LIN {X 0,Y 361.187,Z 795.351,A -85,B 0,C 180,E1 -13387.357,E2 -13387.357} C_VEL
LIN {X 0,Y 363.65,Z 828.384,A -85,B 0,C 180,E1 -13388.543,E2 -13388.543} C_VEL
LIN {X 0,Y 361.748,Z 885.155,A -85,B 0,C 180,E1 -13390.011,E2 -13390.011} C_VEL
LIN {X 0,Y 361.085,Z 897.459,A -85,B 0,C 180,E1 -13390.491,E2 -13390.491} C_VEL
LIN {X 0,Y 360.263,Z 910.027,A -85,B 0,C 180,E1 -13391.074,E2 -13391.074} C_VEL
LIN {X 0,Y 359.139,Z 922.712,A -85,B 0,C 180,E1 -13391.9,E2 -13391.9} C_VEL
LIN {X 0,Y 357.978,Z 934.051,A -85,B 0,C 180,E1 -13392.872,E2 -13392.872} C_VEL
LIN {X 0,Y 356.772,Z 945.633,A -85,B 0,C 180,E1 -13394.136,E2 -13394.136} C_VEL
LIN {X 0,Y 355.868,Z 954.88,A -85,B 0,C 180,E1 -13395.397,E2 -13395.397} C_VEL
LIN {X 0,Y 355.115,Z 963.565,A -85,B 0,C 180,E1 -13396.843,E2 -13396.843} C_VEL
LIN {X 0,Y 354.408,Z 971.955,A -85,B 0,C 180,E1 -13398.561,E2 -13398.561} C_VEL
LIN {X 0,Y 354.031,Z 978.739,A -85,B 0,C 180,E1 -13400.284,E2 -13400.284} C_VEL
LIN {X 0,Y 353.925,Z 984.165,A -85,B 0,C 180,E1 -13402.008,E2 -13402.008} C_VEL
LIN {X 0,Y 353.966,Z 987.855,A -85,B 0,C 180,E1 -13403.493,E2 -13403.493} C_VEL
LIN {X 0,Y 354.122,Z 991.509,A -85,B 0,C 180,E1 -13405.445,E2 -13405.445} C_VEL
LIN {X 0,Y 354.197,Z 993.033,A -85,B 0,C 180,E1 -13406.586,E2 -13406.586} C_VEL
LIN {X 0,Y 354.246,Z 994.085,A -85,B 0,C 180,E1 -13407.724,E2 -13407.724} C_VEL
LIN {X 0,Y 354.313,Z 994.729,A -85,B 0,C 180,E1 -13408.862,E2 -13408.862} C_VEL
LIN {X 0,Y 354.371,Z 994.965,A -85,B 0,C 180,E1 -13409.998,E2 -13409.998} C_VEL
LIN {X 0,Y 354.307,Z 994.762,A -85,B 0,C 180,E1 -13411.135,E2 -13411.135} C_VEL
LIN {X 0,Y 354.238,Z 994.109,A -85,B 0,C 180,E1 -13412.272,E2 -13412.272} C_VEL
LIN {X 0,Y 354.193,Z 993.052,A -85,B 0,C 180,E1 -13413.411,E2 -13413.411} C_VEL
LIN {X 0,Y 354.116,Z 991.578,A -85,B 0,C 180,E1 -13414.552,E2 -13414.552} C_VEL
LIN {X 0,Y 353.962,Z 987.944,A -85,B 0,C 180,E1 -13416.533,E2 -13416.533} C_VEL
LIN {X 0,Y 353.921,Z 982.715,A -85,B 0,C 180,E1 -13418.563,E2 -13418.563} C_VEL
LIN {X 0,Y 354.153,Z 975.942,A -85,B 0,C 180,E1 -13420.575,E2 -13420.575} C_VEL
LIN {X 0,Y 354.69,Z 968.615,A -85,B 0,C 180,E1 -13422.297,E2 -13422.297} C_VEL
LIN {X 0,Y 355.571,Z 960.085,A -85,B 0,C 180,E1 -13423.915,E2 -13423.915} C_VEL
LIN {X 0,Y 356.435,Z 951.284,A -85,B 0,C 180,E1 -13425.289,E2 -13425.289} C_VEL
LIN {X 0,Y 357.256,Z 942.549,A -85,B 0,C 180,E1 -13426.425,E2 -13426.425} C_VEL
LIN {X 0,Y 358.722,Z 930.579,A -85,B 0,C 180,E1 -13427.676,E2 -13427.676} C_VEL
LIN {X 0,Y 359.936,Z 918.59,A -85,B 0,C 180,E1 -13428.645,E2 -13428.645} C_VEL
LIN {X 0,Y 361.04,Z 906.197,A -85,B 0,C 180,E1 -13429.397,E2 -13429.397} C_VEL
LIN {X 0,Y 361.965,Z 892.632,A -85,B 0,C 180,E1 -13429.973,E2 -13429.973} C_VEL
LIN {X 0,Y 362.399,Z 877.372,A -85,B 0,C 180,E1 -13430.355,E2 -13430.355} C_VEL
LIN {X 0,Y 363.215,Z 826.987,A -85,B 0,C 180,E1 -13431.38,E2 -13431.38} C_VEL
LIN {X 0,Y 359.888,Z 793.813,A -85,B 0,C 180,E1 -13432.316,E2 -13432.316} C_VEL
LIN {X 0,Y 357.689,Z 776.377,A -85,B 0,C 180,E1 -13432.881,E2 -13432.881} C_VEL
LIN {X 0,Y 359.216,Z 759.596,A -85,B 0,C 180,E1 -13435.844,E2 -13435.844} C_VEL
LIN {X 0,Y 361.25,Z 739.879,A -85,B 0,C 180,E1 -13439.419,E2 -13439.419} C_VEL
LIN {X 0,Y 361.354,Z 736.535,A -85,B 0,C 180,E1 -13440.052,E2 -13440.052} C_VEL
LIN {X 0,Y 358.531,Z 723.308,A -85,B 0,C 180,E1 -13442.85,E2 -13442.85} C_VEL
LIN {X 0,Y 355.677,Z 711.544,A -85,B 0,C 180,E1 -13445.502,E2 -13445.502} C_VEL
LIN {X 0,Y 354.855,Z 708.388,A -85,B 0,C 180,E1 -13446.295,E2 -13446.295} C_VEL
LIN {X 0,Y 354.817,Z 708.289,A -85,B 0,C 180,E1 -13449.422,E2 -13449.422} C_VEL
LIN {X 0,Y 354.781,Z 708.286,A -85,B 0,C 180,E1 -13452.866,E2 -13452.866} C_VEL
LIN {X 0,Y 354.761,Z 708.286,A -85,B 0,C 180,E1 -13456.103,E2 -13456.103} C_VEL
LIN {X 0,Y 354.78,Z 708.284,A -85,B 0,C 180,E1 -13459.178,E2 -13459.178} C_VEL
LIN {X 0,Y 354.803,Z 708.289,A -85,B 0,C 180,E1 -13462.4,E2 -13462.4} C_VEL
LIN {X 0,Y 354.802,Z 708.275,A -85,B 0,C 180,E1 -13464.94,E2 -13464.94} C_VEL
LIN {X 0,Y 354.783,Z 708.289,A -85,B 0,C 180,E1 -13468.404,E2 -13468.404} C_VEL
LIN {X 0,Y 354.843,Z 708.281,A -85,B 0,C 180,E1 -13471.618,E2 -13471.618} C_VEL
LIN {X 0,Y 354.888,Z 708.275,A -85,B 0,C 180,E1 -13474.172,E2 -13474.172} C_VEL
LIN {X 0,Y 354.823,Z 708.282,A -85,B 0,C 180,E1 -13477.893,E2 -13477.893} C_VEL
LIN {X 0,Y 354.911,Z 708.27,A -85,B 0,C 180,E1 -13481.891,E2 -13481.891} C_VEL
LIN {X 0,Y 354.931,Z 708.268,A -85,B 0,C 180,E1 -13485.981,E2 -13485.981} C_VEL
LIN {X 0,Y 354.966,Z 708.269,A -85,B 0,C 180,E1 -13489.736,E2 -13489.736} C_VEL
LIN {X 0,Y 355.112,Z 708.248,A -85,B 0,C 180,E1 -13493.18,E2 -13493.18} C_VEL
LIN {X 0,Y 355.234,Z 708.233,A -85,B 0,C 180,E1 -13497.732,E2 -13497.732} C_VEL
LIN {X 0,Y 355.385,Z 708.21,A -85,B 0,C 180,E1 -13500,E2 -13500} C_VEL
LIN {X 0,Y 355.233,Z 708.236,A -85,B 0,C 180,E1 -13502.268,E2 -13502.268} C_VEL
LIN {X 0,Y 355.125,Z 708.249,A -85,B 0,C 180,E1 -13506.82,E2 -13506.82} C_VEL
LIN {X 0,Y 355.004,Z 708.26,A -85,B 0,C 180,E1 -13509.113,E2 -13509.113} C_VEL
LIN {X 0,Y 354.91,Z 708.271,A -85,B 0,C 180,E1 -13512.582,E2 -13512.582} C_VEL
LIN {X 0,Y 354.878,Z 708.272,A -85,B 0,C 180,E1 -13516.097,E2 -13516.097} C_VEL
LIN {X 0,Y 354.89,Z 708.278,A -85,B 0,C 180,E1 -13518.473,E2 -13518.473} C_VEL
LIN {X 0,Y 354.804,Z 708.283,A -85,B 0,C 180,E1 -13522.108,E2 -13522.108} C_VEL
LIN {X 0,Y 354.887,Z 708.281,A -85,B 0,C 180,E1 -13525.829,E2 -13525.829} C_VEL
LIN {X 0,Y 354.808,Z 708.284,A -85,B 0,C 180,E1 -13529.683,E2 -13529.683} C_VEL
LIN {X 0,Y 354.797,Z 708.286,A -85,B 0,C 180,E1 -13533.703,E2 -13533.703} C_VEL
LIN {X 0,Y 354.793,Z 708.285,A -85,B 0,C 180,E1 -13536.461,E2 -13536.461} C_VEL
LIN {X 0,Y 354.816,Z 708.285,A -85,B 0,C 180,E1 -13539.425,E2 -13539.425} C_VEL
LIN {X 0,Y 354.839,Z 708.428,A -85,B 0,C 180,E1 -13542.292,E2 -13542.292} C_VEL
LIN {X 0,Y 355.063,Z 709.428,A -85,B 0,C 180,E1 -13542.499,E2 -13542.499} C_VEL
LIN {X 0,Y 361.993,Z 724.642,A -85,B 0,C 180,E1 -13543.378,E2 -13543.378} C_VEL
LIN {X 0,Y 364.783,Z 731.44,A -85,B 0,C 180,E1 -13543.724,E2 -13543.724} C_VEL
LIN {X 0,Y 363.92,Z 784.743,A -85,B 0,C 180,E1 -13544.825,E2 -13544.825} C_VEL
LIN {X 0,Y 363.875,Z 798.11,A -85,B 0,C 180,E1 -13545.213,E2 -13545.213} C_VEL
LIN {X 0,Y 363.637,Z 810.174,A -85,B 0,C 180,E1 -13545.778,E2 -13545.778} C_VEL
LIN {X 0,Y 363.079,Z 822.796,A -85,B 0,C 180,E1 -13546.597,E2 -13546.597} C_VEL
LIN {X 0,Y 362.232,Z 834.729,A -85,B 0,C 180,E1 -13547.626,E2 -13547.626} C_VEL
LIN {X 0,Y 361.284,Z 845.818,A -85,B 0,C 180,E1 -13548.858,E2 -13548.858} C_VEL
LIN {X 0,Y 360.216,Z 856.083,A -85,B 0,C 180,E1 -13550.288,E2 -13550.288} C_VEL
LIN {X 0,Y 359.068,Z 865.467,A -85,B 0,C 180,E1 -13551.938,E2 -13551.938} C_VEL
LIN {X 0,Y 358.091,Z 872.957,A -85,B 0,C 180,E1 -13553.58,E2 -13553.58} C_VEL
LIN {X 0,Y 357.329,Z 878.96,A -85,B 0,C 180,E1 -13555.226,E2 -13555.226} C_VEL
LIN {X 0,Y 356.46,Z 884.482,A -85,B 0,C 180,E1 -13557.169,E2 -13557.169} C_VEL
LIN {X 0,Y 355.92,Z 888.534,A -85,B 0,C 180,E1 -13559.112,E2 -13559.112} C_VEL
LIN {X 0,Y 355.612,Z 890.545,A -85,B 0,C 180,E1 -13560.41,E2 -13560.41} C_VEL
LIN {X 0,Y 355.379,Z 891.923,A -85,B 0,C 180,E1 -13561.667,E2 -13561.667} C_VEL
LIN {X 0,Y 355.21,Z 892.853,A -85,B 0,C 180,E1 -13562.933,E2 -13562.933} C_VEL
LIN {X 0,Y 355.1,Z 893.271,A -85,B 0,C 180,E1 -13564.19,E2 -13564.19} C_VEL
LIN {X 0,Y 355.01,Z 893.189,A -85,B 0,C 180,E1 -13565.596,E2 -13565.596} C_VEL
LIN {X 0,Y 355.031,Z 892.728,A -85,B 0,C 180,E1 -13566.679,E2 -13566.679} C_VEL
LIN {X 0,Y 355.205,Z 891.198,A -85,B 0,C 180,E1 -13568.425,E2 -13568.425} C_VEL
LIN {X 0,Y 355.566,Z 888.364,A -85,B 0,C 180,E1 -13570.368,E2 -13570.368} C_VEL
LIN {X 0,Y 356.038,Z 884.542,A -85,B 0,C 180,E1 -13572.186,E2 -13572.186} C_VEL
LIN {X 0,Y 356.602,Z 879.534,A -85,B 0,C 180,E1 -13573.985,E2 -13573.985} C_VEL
LIN {X 0,Y 357.322,Z 873.189,A -85,B 0,C 180,E1 -13575.769,E2 -13575.769} C_VEL
LIN {X 0,Y 358.214,Z 865.265,A -85,B 0,C 180,E1 -13577.538,E2 -13577.538} C_VEL
LIN {X 0,Y 359.042,Z 857.126,A -85,B 0,C 180,E1 -13578.999,E2 -13578.999} C_VEL
LIN {X 0,Y 359.999,Z 847.172,A -85,B 0,C 180,E1 -13580.45,E2 -13580.45} C_VEL
LIN {X 0,Y 360.918,Z 836.089,A -85,B 0,C 180,E1 -13581.745,E2 -13581.745} C_VEL
LIN {X 0,Y 361.715,Z 824.779,A -85,B 0,C 180,E1 -13582.779,E2 -13582.779} C_VEL
LIN {X 0,Y 362.31,Z 812.227,A -85,B 0,C 180,E1 -13583.668,E2 -13583.668} C_VEL
LIN {X 0,Y 362.675,Z 799.879,A -85,B 0,C 180,E1 -13584.302,E2 -13584.302} C_VEL
LIN {X 0,Y 362.785,Z 787.742,A -85,B 0,C 180,E1 -13584.717,E2 -13584.717} C_VEL
LIN {X 0,Y 363.57,Z 731.522,A -85,B 0,C 180,E1 -13585.873,E2 -13585.873} C_VEL
LIN {X 0,Y 363.342,Z 729.011,A -85,B 0,C 180,E1 -13585.94,E2 -13585.94} C_VEL
LIN {X 0,Y 355.205,Z 709.198,A -85,B 0,C 180,E1 -13586.883,E2 -13586.883} C_VEL
LIN {X 0,Y 355.09,Z 708.341,A -85,B 0,C 180,E1 -13587.095,E2 -13587.095} C_VEL
LIN {X 0,Y 355.148,Z 708.249,A -85,B 0,C 180,E1 -13588.868,E2 -13588.868} C_VEL
LIN {X 0,Y 355.222,Z 708.236,A -85,B 0,C 180,E1 -13592.269,E2 -13592.269} C_VEL
LIN {X 0,Y 355.089,Z 708.249,A -85,B 0,C 180,E1 -13596.822,E2 -13596.822} C_VEL
LIN {X 0,Y 354.955,Z 708.265,A -85,B 0,C 180,E1 -13600.266,E2 -13600.266} C_VEL
LIN {X 0,Y 354.948,Z 708.267,A -85,B 0,C 180,E1 -13604.02,E2 -13604.02} C_VEL
LIN {X 0,Y 354.872,Z 708.279,A -85,B 0,C 180,E1 -13607.518,E2 -13607.518} C_VEL
LIN {X 0,Y 354.823,Z 708.283,A -85,B 0,C 180,E1 -13611.418,E2 -13611.418} C_VEL
LIN {X 0,Y 354.794,Z 708.285,A -85,B 0,C 180,E1 -13612.45,E2 -13612.45} C_VEL
LIN {X 0,Y 354.118,Z 708.375,A -85,B 0,C 180,E1 -13613.396,E2 -13613.396} C_VEL
LIN {X 0,Y 351.283,Z 708.719,A -85,B 0,C 180,E1 -13614.937,E2 -13614.937} C_VEL
LIN {X 0,Y 348.879,Z 709.01,A -85,B 0,C 180,E1 -13616.183,E2 -13616.183} C_VEL
LIN {X 0,Y 347.832,Z 709.14,A -85,B 0,C 180,E1 -13617.147,E2 -13617.147} C_VEL
LIN {X 0,Y 347.738,Z 709.155,A -85,B 0,C 180,E1 -13617.473,E2 -13617.473} C_VEL
LIN {X 0,Y 347.736,Z 709.167,A -85,B 0,C 180,E1 -13620.351,E2 -13620.351} C_VEL
LIN {X 0,Y 347.755,Z 709.143,A -85,B 0,C 180,E1 -13624.045,E2 -13624.045} C_VEL
LIN {X 0,Y 347.76,Z 709.155,A -85,B 0,C 180,E1 -13627.323,E2 -13627.323} C_VEL
LIN {X 0,Y 347.702,Z 709.171,A -85,B 0,C 180,E1 -13630.303,E2 -13630.303} C_VEL
LIN {X 0,Y 347.72,Z 709.173,A -85,B 0,C 180,E1 -13633.411,E2 -13633.411} C_VEL
LIN {X 0,Y 347.728,Z 709.168,A -85,B 0,C 180,E1 -13636.688,E2 -13636.688} C_VEL
LIN {X 0,Y 347.708,Z 709.174,A -85,B 0,C 180,E1 -13640.183,E2 -13640.183} C_VEL
LIN {X 0,Y 347.76,Z 709.166,A -85,B 0,C 180,E1 -13642.678,E2 -13642.678} C_VEL
LIN {X 0,Y 347.857,Z 709.393,A -85,B 0,C 180,E1 -13645.736,E2 -13645.736} C_VEL
LIN {X 0,Y 348.03,Z 710.197,A -85,B 0,C 180,E1 -13645.89,E2 -13645.89} C_VEL
LIN {X 0,Y 354.796,Z 729.357,A -85,B 0,C 180,E1 -13646.733,E2 -13646.733} C_VEL
LIN {X 0,Y 353.601,Z 786.373,A -85,B 0,C 180,E1 -13648.146,E2 -13648.146} C_VEL
LIN {X 0,Y 353.411,Z 797.802,A -85,B 0,C 180,E1 -13648.596,E2 -13648.596} C_VEL
LIN {X 0,Y 353.102,Z 808.375,A -85,B 0,C 180,E1 -13649.168,E2 -13649.168} C_VEL
LIN {X 0,Y 352.703,Z 817.545,A -85,B 0,C 180,E1 -13649.792,E2 -13649.792} C_VEL
LIN {X 0,Y 352.091,Z 828.422,A -85,B 0,C 180,E1 -13650.722,E2 -13650.722} C_VEL
LIN {X 0,Y 351.487,Z 837.924,A -85,B 0,C 180,E1 -13651.72,E2 -13651.72} C_VEL
LIN {X 0,Y 350.886,Z 846.039,A -85,B 0,C 180,E1 -13652.731,E2 -13652.731} C_VEL
LIN {X 0,Y 350.414,Z 853.461,A -85,B 0,C 180,E1 -13653.817,E2 -13653.817} C_VEL
LIN {X 0,Y 349.887,Z 860.653,A -85,B 0,C 180,E1 -13655.05,E2 -13655.05} C_VEL
LIN {X 0,Y 349.234,Z 868.074,A -85,B 0,C 180,E1 -13656.581,E2 -13656.581} C_VEL
LIN {X 0,Y 348.791,Z 873.676,A -85,B 0,C 180,E1 -13657.957,E2 -13657.957} C_VEL
LIN {X 0,Y 348.471,Z 878.376,A -85,B 0,C 180,E1 -13659.332,E2 -13659.332} C_VEL
LIN {X 0,Y 348.153,Z 883.303,A -85,B 0,C 180,E1 -13661.156,E2 -13661.156} C_VEL
LIN {X 0,Y 347.914,Z 886.997,A -85,B 0,C 180,E1 -13662.968,E2 -13662.968} C_VEL
LIN {X 0,Y 347.775,Z 889.586,A -85,B 0,C 180,E1 -13664.769,E2 -13664.769} C_VEL
LIN {X 0,Y 347.82,Z 890.797,A -85,B 0,C 180,E1 -13665.967,E2 -13665.967} C_VEL
LIN {X 0,Y 347.854,Z 891.478,A -85,B 0,C 180,E1 -13667.159,E2 -13667.159} C_VEL
LIN {X 0,Y 347.981,Z 891.721,A -85,B 0,C 180,E1 -13668.348,E2 -13668.348} C_VEL
LIN {X 0,Y 348.178,Z 891.547,A -85,B 0,C 180,E1 -13669.533,E2 -13669.533} C_VEL
LIN {X 0,Y 348.509,Z 890.537,A -85,B 0,C 180,E1 -13671.172,E2 -13671.172} C_VEL
LIN {X 0,Y 349.011,Z 888.328,A -85,B 0,C 180,E1 -13673.06,E2 -13673.06} C_VEL
LIN {X 0,Y 349.623,Z 885.176,A -85,B 0,C 180,E1 -13674.81,E2 -13674.81} C_VEL
LIN {X 0,Y 350.327,Z 880.893,A -85,B 0,C 180,E1 -13676.549,E2 -13676.549} C_VEL
LIN {X 0,Y 351.132,Z 875.354,A -85,B 0,C 180,E1 -13678.279,E2 -13678.279} C_VEL
LIN {X 0,Y 352.021,Z 870.096,A -85,B 0,C 180,E1 -13679.62,E2 -13679.62} C_VEL
LIN {X 0,Y 353.034,Z 862.825,A -85,B 0,C 180,E1 -13681.141,E2 -13681.141} C_VEL
LIN {X 0,Y 353.898,Z 856.366,A -85,B 0,C 180,E1 -13682.276,E2 -13682.276} C_VEL
LIN {X 0,Y 354.886,Z 847.639,A -85,B 0,C 180,E1 -13683.548,E2 -13683.548} C_VEL
LIN {X 0,Y 355.855,Z 838.207,A -85,B 0,C 180,E1 -13684.673,E2 -13684.673} C_VEL
LIN {X 0,Y 356.553,Z 829.764,A -85,B 0,C 180,E1 -13685.514,E2 -13685.514} C_VEL
LIN {X 0,Y 357.209,Z 819.421,A -85,B 0,C 180,E1 -13686.354,E2 -13686.354} C_VEL
LIN {X 0,Y 357.742,Z 809.048,A -85,B 0,C 180,E1 -13687.017,E2 -13687.017} C_VEL
LIN {X 0,Y 358.112,Z 798.99,A -85,B 0,C 180,E1 -13687.506,E2 -13687.506} C_VEL
LIN {X 0,Y 358.317,Z 785.894,A -85,B 0,C 180,E1 -13687.959,E2 -13687.959} C_VEL
LIN {X 0,Y 359.291,Z 754.548,A -85,B 0,C 180,E1 -13688.813,E2 -13688.813} C_VEL
LIN {X 0,Y 360.134,Z 733.434,A -85,B 0,C 180,E1 -13689.39,E2 -13689.39} C_VEL
LIN {X 0,Y 354.89,Z 722.496,A -85,B 0,C 180,E1 -13690.29,E2 -13690.29} C_VEL
LIN {X 0,Y 349.346,Z 712.616,A -85,B 0,C 180,E1 -13691.263,E2 -13691.263} C_VEL
LIN {X 0,Y 347.986,Z 709.706,A -85,B 0,C 180,E1 -13691.585,E2 -13691.585} C_VEL
LIN {X 0,Y 347.883,Z 709.168,A -85,B 0,C 180,E1 -13691.951,E2 -13691.951} C_VEL
LIN {X 0,Y 347.872,Z 709.153,A -85,B 0,C 180,E1 -13695.226,E2 -13695.226} C_VEL
LIN {X 0,Y 347.81,Z 709.161,A -85,B 0,C 180,E1 -13698.863,E2 -13698.863} C_VEL
LIN {X 0,Y 347.769,Z 709.168,A -85,B 0,C 180,E1 -13702.58,E2 -13702.58} C_VEL
LIN {X 0,Y 347.8,Z 709.161,A -85,B 0,C 180,E1 -13705.109,E2 -13705.109} C_VEL
LIN {X 0,Y 347.764,Z 709.166,A -85,B 0,C 180,E1 -13709.014,E2 -13709.014} C_VEL
LIN {X 0,Y 347.74,Z 709.17,A -85,B 0,C 180,E1 -13713.071,E2 -13713.071} C_VEL
LIN {X 0,Y 347.777,Z 709.164,A -85,B 0,C 180,E1 -13716.064,E2 -13716.064} C_VEL
LIN {X 0,Y 347.759,Z 709.165,A -85,B 0,C 180,E1 -13718.792,E2 -13718.792} C_VEL
LIN {X 0,Y 347.757,Z 709.168,A -85,B 0,C 180,E1 -13721.829,E2 -13721.829} C_VEL
LIN {X 0,Y 347.712,Z 709.171,A -85,B 0,C 180,E1 -13725.026,E2 -13725.026} C_VEL
LIN {X 0,Y 347.756,Z 709.167,A -85,B 0,C 180,E1 -13728.396,E2 -13728.396} C_VEL
LIN {X 0,Y 347.778,Z 709.165,A -85,B 0,C 180,E1 -13732.01,E2 -13732.01} C_VEL
LIN {X 0,Y 347.815,Z 709.357,A -85,B 0,C 180,E1 -13733.781,E2 -13733.781} C_VEL
LIN {X 0,Y 351.296,Z 723.703,A -85,B 0,C 180,E1 -13736.963,E2 -13736.963} C_VEL
LIN {X 0,Y 354.079,Z 736.282,A -85,B 0,C 180,E1 -13739.591,E2 -13739.591} C_VEL
LIN {X 0,Y 354.337,Z 739.773,A -85,B 0,C 180,E1 -13740.272,E2 -13740.272} C_VEL
LIN {X 0,Y 352.046,Z 761.67,A -85,B 0,C 180,E1 -13744.264,E2 -13744.264} C_VEL
LIN {X 0,Y 351.359,Z 769.237,A -85,B 0,C 180,E1 -13745.572,E2 -13745.572} C_VEL
LIN {X 0,Y 354.075,Z 789.134,A -85,B 0,C 180,E1 -13746.512,E2 -13746.512} C_VEL
LIN {X 0,Y 355.43,Z 801.877,A -85,B 0,C 180,E1 -13747.047,E2 -13747.047} C_VEL
LIN {X 0,Y 357.266,Z 829.438,A -85,B 0,C 180,E1 -13748.051,E2 -13748.051} C_VEL
LIN {X 0,Y 355.318,Z 884.018,A -85,B 0,C 180,E1 -13749.52,E2 -13749.52} C_VEL
LIN {X 0,Y 354.697,Z 894.667,A -85,B 0,C 180,E1 -13749.937,E2 -13749.937} C_VEL
LIN {X 0,Y 353.755,Z 906.444,A -85,B 0,C 180,E1 -13750.561,E2 -13750.561} C_VEL
LIN {X 0,Y 352.389,Z 921.354,A -85,B 0,C 180,E1 -13751.54,E2 -13751.54} C_VEL
LIN {X 0,Y 351.173,Z 932.777,A -85,B 0,C 180,E1 -13752.529,E2 -13752.529} C_VEL
LIN {X 0,Y 350.055,Z 943.219,A -85,B 0,C 180,E1 -13753.674,E2 -13753.674} C_VEL
LIN {X 0,Y 349.023,Z 953.3,A -85,B 0,C 180,E1 -13755.043,E2 -13755.043} C_VEL
LIN {X 0,Y 348.18,Z 962.42,A -85,B 0,C 180,E1 -13756.576,E2 -13756.576} C_VEL
LIN {X 0,Y 347.404,Z 970.83,A -85,B 0,C 180,E1 -13758.327,E2 -13758.327} C_VEL
LIN {X 0,Y 346.999,Z 977.635,A -85,B 0,C 180,E1 -13760.085,E2 -13760.085} C_VEL
LIN {X 0,Y 346.862,Z 983.078,A -85,B 0,C 180,E1 -13761.844,E2 -13761.844} C_VEL
LIN {X 0,Y 346.919,Z 986.997,A -85,B 0,C 180,E1 -13763.454,E2 -13763.454} C_VEL
LIN {X 0,Y 347.062,Z 990.46,A -85,B 0,C 180,E1 -13765.352,E2 -13765.352} C_VEL
LIN {X 0,Y 347.152,Z 991.999,A -85,B 0,C 180,E1 -13766.516,E2 -13766.516} C_VEL
LIN {X 0,Y 347.205,Z 993.06,A -85,B 0,C 180,E1 -13767.678,E2 -13767.678} C_VEL
LIN {X 0,Y 347.279,Z 993.711,A -85,B 0,C 180,E1 -13768.839,E2 -13768.839} C_VEL
LIN {X 0,Y 347.343,Z 993.953,A -85,B 0,C 180,E1 -13769.998,E2 -13769.998} C_VEL
LIN {X 0,Y 347.271,Z 993.758,A -85,B 0,C 180,E1 -13771.158,E2 -13771.158} C_VEL
LIN {X 0,Y 347.195,Z 993.11,A -85,B 0,C 180,E1 -13772.318,E2 -13772.318} C_VEL
LIN {X 0,Y 347.148,Z 992.057,A -85,B 0,C 180,E1 -13773.48,E2 -13773.48} C_VEL
LIN {X 0,Y 347.056,Z 990.583,A -85,B 0,C 180,E1 -13774.644,E2 -13774.644} C_VEL
LIN {X 0,Y 346.919,Z 987.211,A -85,B 0,C 180,E1 -13776.546,E2 -13776.546} C_VEL
LIN {X 0,Y 346.833,Z 983.37,A -85,B 0,C 180,E1 -13778.153,E2 -13778.153} C_VEL
LIN {X 0,Y 347.009,Z 977.097,A -85,B 0,C 180,E1 -13780.206,E2 -13780.206} C_VEL
LIN {X 0,Y 347.493,Z 970.264,A -85,B 0,C 180,E1 -13781.963,E2 -13781.963} C_VEL
LIN {X 0,Y 348.159,Z 963.381,A -85,B 0,C 180,E1 -13783.421,E2 -13783.421} C_VEL
LIN {X 0,Y 349.045,Z 954.52,A -85,B 0,C 180,E1 -13784.972,E2 -13784.972} C_VEL
LIN {X 0,Y 350.158,Z 944.035,A -85,B 0,C 180,E1 -13786.467,E2 -13786.467} C_VEL
LIN {X 0,Y 351.575,Z 932.67,A -85,B 0,C 180,E1 -13787.747,E2 -13787.747} C_VEL
LIN {X 0,Y 352.811,Z 921.592,A -85,B 0,C 180,E1 -13788.734,E2 -13788.734} C_VEL
LIN {X 0,Y 354.056,Z 909.409,A -85,B 0,C 180,E1 -13789.569,E2 -13789.569} C_VEL
LIN {X 0,Y 355.016,Z 896.926,A -85,B 0,C 180,E1 -13790.192,E2 -13790.192} C_VEL
LIN {X 0,Y 355.654,Z 884.128,A -85,B 0,C 180,E1 -13790.607,E2 -13790.607} C_VEL
LIN {X 0,Y 356.612,Z 827.527,A -85,B 0,C 180,E1 -13791.794,E2 -13791.794} C_VEL
LIN {X 0,Y 353.362,Z 794.632,A -85,B 0,C 180,E1 -13792.743,E2 -13792.743} C_VEL
LIN {X 0,Y 350.889,Z 775.382,A -85,B 0,C 180,E1 -13793.376,E2 -13793.376} C_VEL
LIN {X 0,Y 352.424,Z 759.116,A -85,B 0,C 180,E1 -13796.306,E2 -13796.306} C_VEL
LIN {X 0,Y 354.45,Z 740.741,A -85,B 0,C 180,E1 -13799.714,E2 -13799.714} C_VEL
LIN {X 0,Y 354.373,Z 737.386,A -85,B 0,C 180,E1 -13800.377,E2 -13800.377} C_VEL
LIN {X 0,Y 351.589,Z 724.466,A -85,B 0,C 180,E1 -13803.186,E2 -13803.186} C_VEL
LIN {X 0,Y 348.899,Z 713.443,A -85,B 0,C 180,E1 -13805.741,E2 -13805.741} C_VEL
LIN {X 0,Y 347.799,Z 709.247,A -85,B 0,C 180,E1 -13806.824,E2 -13806.824} C_VEL
LIN {X 0,Y 347.725,Z 709.167,A -85,B 0,C 180,E1 -13810.295,E2 -13810.295} C_VEL
LIN {X 0,Y 347.719,Z 709.166,A -85,B 0,C 180,E1 -13813.406,E2 -13813.406} C_VEL
LIN {X 0,Y 347.717,Z 709.164,A -85,B 0,C 180,E1 -13816.685,E2 -13816.685} C_VEL
LIN {X 0,Y 347.738,Z 709.156,A -85,B 0,C 180,E1 -13820.172,E2 -13820.172} C_VEL
LIN {X 0,Y 347.756,Z 709.169,A -85,B 0,C 180,E1 -13822.679,E2 -13822.679} C_VEL
LIN {X 0,Y 347.738,Z 709.165,A -85,B 0,C 180,E1 -13825.955,E2 -13825.955} C_VEL
LIN {X 0,Y 347.754,Z 709.169,A -85,B 0,C 180,E1 -13829.653,E2 -13829.653} C_VEL
LIN {X 0,Y 347.842,Z 709.153,A -85,B 0,C 180,E1 -13832.743,E2 -13832.743} C_VEL
LIN {X 0,Y 347.777,Z 709.163,A -85,B 0,C 180,E1 -13836.161,E2 -13836.161} C_VEL
LIN {X 0,Y 347.806,Z 709.161,A -85,B 0,C 180,E1 -13839.909,E2 -13839.909} C_VEL
LIN {X 0,Y 347.855,Z 709.146,A -85,B 0,C 180,E1 -13842.359,E2 -13842.359} C_VEL
LIN {X 0,Y 347.885,Z 709.145,A -85,B 0,C 180,E1 -13845.97,E2 -13845.97} C_VEL
LIN {X 0,Y 347.916,Z 709.147,A -85,B 0,C 180,E1 -13849.525,E2 -13849.525} C_VEL
LIN {X 0,Y 348.078,Z 709.125,A -85,B 0,C 180,E1 -13853.042,E2 -13853.042} C_VEL
LIN {X 0,Y 348.197,Z 709.109,A -85,B 0,C 180,E1 -13857.687,E2 -13857.687} C_VEL
LIN {X 0,Y 348.334,Z 709.088,A -85,B 0,C 180,E1 -13860,E2 -13860} C_VEL
LIN {X 0,Y 348.196,Z 709.113,A -85,B 0,C 180,E1 -13862.314,E2 -13862.314} C_VEL
LIN {X 0,Y 348.093,Z 709.124,A -85,B 0,C 180,E1 -13866.958,E2 -13866.958} C_VEL
LIN {X 0,Y 347.956,Z 709.139,A -85,B 0,C 180,E1 -13869.299,E2 -13869.299} C_VEL
LIN {X 0,Y 347.879,Z 709.147,A -85,B 0,C 180,E1 -13872.84,E2 -13872.84} C_VEL
LIN {X 0,Y 347.827,Z 709.151,A -85,B 0,C 180,E1 -13876.432,E2 -13876.432} C_VEL
LIN {X 0,Y 347.839,Z 709.154,A -85,B 0,C 180,E1 -13878.861,E2 -13878.861} C_VEL
LIN {X 0,Y 347.751,Z 709.156,A -85,B 0,C 180,E1 -13882.581,E2 -13882.581} C_VEL
LIN {X 0,Y 347.8,Z 709.155,A -85,B 0,C 180,E1 -13885.11,E2 -13885.11} C_VEL
LIN {X 0,Y 347.798,Z 709.152,A -85,B 0,C 180,E1 -13887.695,E2 -13887.695} C_VEL
LIN {X 0,Y 347.74,Z 709.171,A -85,B 0,C 180,E1 -13890.349,E2 -13890.349} C_VEL
LIN {X 0,Y 347.739,Z 709.17,A -85,B 0,C 180,E1 -13894.045,E2 -13894.045} C_VEL
LIN {X 0,Y 347.758,Z 709.168,A -85,B 0,C 180,E1 -13897.322,E2 -13897.322} C_VEL
LIN {X 0,Y 347.725,Z 709.172,A -85,B 0,C 180,E1 -13900.298,E2 -13900.298} C_VEL
LIN {X 0,Y 347.786,Z 709.337,A -85,B 0,C 180,E1 -13901.769,E2 -13901.769} C_VEL
LIN {X 0,Y 348.057,Z 710.428,A -85,B 0,C 180,E1 -13901.98,E2 -13901.98} C_VEL
LIN {X 0,Y 355.106,Z 725.654,A -85,B 0,C 180,E1 -13902.897,E2 -13902.897} C_VEL
LIN {X 0,Y 358.261,Z 732.986,A -85,B 0,C 180,E1 -13903.294,E2 -13903.294} C_VEL
LIN {X 0,Y 357.367,Z 788.959,A -85,B 0,C 180,E1 -13904.483,E2 -13904.483} C_VEL
LIN {X 0,Y 357.262,Z 802.328,A -85,B 0,C 180,E1 -13904.935,E2 -13904.935} C_VEL
LIN {X 0,Y 356.958,Z 814.44,A -85,B 0,C 180,E1 -13905.566,E2 -13905.566} C_VEL
LIN {X 0,Y 356.365,Z 825.612,A -85,B 0,C 180,E1 -13906.353,E2 -13906.353} C_VEL
LIN {X 0,Y 355.424,Z 837.818,A -85,B 0,C 180,E1 -13907.475,E2 -13907.475} C_VEL
LIN {X 0,Y 354.457,Z 848.554,A -85,B 0,C 180,E1 -13908.736,E2 -13908.736} C_VEL
LIN {X 0,Y 353.214,Z 858.923,A -85,B 0,C 180,E1 -13910.27,E2 -13910.27} C_VEL
LIN {X 0,Y 352.198,Z 867.163,A -85,B 0,C 180,E1 -13911.789,E2 -13911.789} C_VEL
LIN {X 0,Y 351.178,Z 874.548,A -85,B 0,C 180,E1 -13913.467,E2 -13913.467} C_VEL
LIN {X 0,Y 350.245,Z 881.069,A -85,B 0,C 180,E1 -13915.357,E2 -13915.357} C_VEL
LIN {X 0,Y 349.473,Z 885.814,A -85,B 0,C 180,E1 -13917.116,E2 -13917.116} C_VEL
LIN {X 0,Y 348.921,Z 889.783,A -85,B 0,C 180,E1 -13919.097,E2 -13919.097} C_VEL
LIN {X 0,Y 348.48,Z 892.453,A -85,B 0,C 180,E1 -13921.054,E2 -13921.054} C_VEL
LIN {X 0,Y 348.239,Z 893.721,A -85,B 0,C 180,E1 -13922.622,E2 -13922.622} C_VEL
LIN {X 0,Y 348.033,Z 894.328,A -85,B 0,C 180,E1 -13924.911,E2 -13924.911} C_VEL
LIN {X 0,Y 347.982,Z 893.979,A -85,B 0,C 180,E1 -13926.178,E2 -13926.178} C_VEL
LIN {X 0,Y 348.171,Z 892.462,A -85,B 0,C 180,E1 -13928.208,E2 -13928.208} C_VEL
LIN {X 0,Y 348.589,Z 889.135,A -85,B 0,C 180,E1 -13930.572,E2 -13930.572} C_VEL
LIN {X 0,Y 349.076,Z 885.239,A -85,B 0,C 180,E1 -13932.424,E2 -13932.424} C_VEL
LIN {X 0,Y 349.7,Z 880.201,A -85,B 0,C 180,E1 -13934.24,E2 -13934.24} C_VEL
LIN {X 0,Y 350.463,Z 873.704,A -85,B 0,C 180,E1 -13936.077,E2 -13936.077} C_VEL
LIN {X 0,Y 351.244,Z 866.967,A -85,B 0,C 180,E1 -13937.61,E2 -13937.61} C_VEL
LIN {X 0,Y 352.092,Z 859.175,A -85,B 0,C 180,E1 -13939.071,E2 -13939.071} C_VEL
LIN {X 0,Y 353.068,Z 849.448,A -85,B 0,C 180,E1 -13940.55,E2 -13940.55} C_VEL
LIN {X 0,Y 354.023,Z 838.649,A -85,B 0,C 180,E1 -13941.87,E2 -13941.87} C_VEL
LIN {X 0,Y 354.844,Z 828.02,A -85,B 0,C 180,E1 -13942.908,E2 -13942.908} C_VEL
LIN {X 0,Y 355.498,Z 815.85,A -85,B 0,C 180,E1 -13943.831,E2 -13943.831} C_VEL
LIN {X 0,Y 355.915,Z 802.681,A -85,B 0,C 180,E1 -13944.566,E2 -13944.566} C_VEL
LIN {X 0,Y 356.105,Z 790.325,A -85,B 0,C 180,E1 -13945.029,E2 -13945.029} C_VEL
LIN {X 0,Y 356.606,Z 744.348,A -85,B 0,C 180,E1 -13946.012,E2 -13946.012} C_VEL
LIN {X 0,Y 356.74,Z 730.81,A -85,B 0,C 180,E1 -13946.297,E2 -13946.297} C_VEL
LIN {X 0,Y 348.227,Z 709.924,A -85,B 0,C 180,E1 -13947.327,E2 -13947.327} C_VEL
LIN {X 0,Y 348.15,Z 709.187,A -85,B 0,C 180,E1 -13947.543,E2 -13947.543} C_VEL
LIN {X 0,Y 348.12,Z 709.122,A -85,B 0,C 180,E1 -13951.159,E2 -13951.159} C_VEL
LIN {X 0,Y 348.184,Z 709.112,A -85,B 0,C 180,E1 -13952.315,E2 -13952.315} C_VEL
LIN {X 0,Y 348.057,Z 709.124,A -85,B 0,C 180,E1 -13956.96,E2 -13956.96} C_VEL
LIN {X 0,Y 347.895,Z 709.144,A -85,B 0,C 180,E1 -13960.477,E2 -13960.477} C_VEL
LIN {X 0,Y 347.905,Z 709.143,A -85,B 0,C 180,E1 -13964.151,E2 -13964.151} C_VEL
LIN {X 0,Y 347.836,Z 709.155,A -85,B 0,C 180,E1 -13967.644,E2 -13967.644} C_VEL
LIN {X 0,Y 347.77,Z 709.162,A -85,B 0,C 180,E1 -13971.626,E2 -13971.626} C_VEL
LIN {X 0,Y 347.744,Z 709.157,A -85,B 0,C 180,E1 -13975.115,E2 -13975.115} C_VEL
LIN {X 0,Y 347.738,Z 709.155,A -85,B 0,C 180,E1 -13977.473,E2 -13977.473} C_VEL
LIN {X 0,Y 347.054,Z 709.251,A -85,B 0,C 180,E1 -13978.44,E2 -13978.44} C_VEL
LIN {X 0,Y 344.219,Z 709.616,A -85,B 0,C 180,E1 -13980.013,E2 -13980.013} C_VEL
LIN {X 0,Y 341.819,Z 709.913,A -85,B 0,C 180,E1 -13981.286,E2 -13981.286} C_VEL
LIN {X 0,Y 340.773,Z 710.032,A -85,B 0,C 180,E1 -13982.27,E2 -13982.27} C_VEL
LIN {X 0,Y 340.678,Z 710.038,A -85,B 0,C 180,E1 -13982.604,E2 -13982.604} C_VEL
LIN {X 0,Y 340.722,Z 710.016,A -85,B 0,C 180,E1 -13985.28,E2 -13985.28} C_VEL
LIN {X 0,Y 340.699,Z 710.041,A -85,B 0,C 180,E1 -13988.383,E2 -13988.383} C_VEL
LIN {X 0,Y 340.671,Z 710.049,A -85,B 0,C 180,E1 -13992.04,E2 -13992.04} C_VEL
LIN {X 0,Y 340.637,Z 710.056,A -85,B 0,C 180,E1 -13995.453,E2 -13995.453} C_VEL
LIN {X 0,Y 340.675,Z 710.047,A -85,B 0,C 180,E1 -13998.688,E2 -13998.688} C_VEL
LIN {X 0,Y 340.724,Z 710.044,A -85,B 0,C 180,E1 -14001.771,E2 -14001.771} C_VEL
LIN {X 0,Y 340.774,Z 710.195,A -85,B 0,C 180,E1 -14005.374,E2 -14005.374} C_VEL
LIN {X 0,Y 340.999,Z 711.108,A -85,B 0,C 180,E1 -14005.568,E2 -14005.568} C_VEL
LIN {X 0,Y 347.987,Z 730.963,A -85,B 0,C 180,E1 -14006.459,E2 -14006.459} C_VEL
LIN {X 0,Y 346.754,Z 786.436,A -85,B 0,C 180,E1 -14007.857,E2 -14007.857} C_VEL
LIN {X 0,Y 346.533,Z 798.8,A -85,B 0,C 180,E1 -14008.351,E2 -14008.351} C_VEL
LIN {X 0,Y 346.187,Z 809.675,A -85,B 0,C 180,E1 -14008.955,E2 -14008.955} C_VEL
LIN {X 0,Y 345.745,Z 819.212,A -85,B 0,C 180,E1 -14009.626,E2 -14009.626} C_VEL
LIN {X 0,Y 345.1,Z 829.968,A -85,B 0,C 180,E1 -14010.573,E2 -14010.573} C_VEL
LIN {X 0,Y 344.526,Z 839.112,A -85,B 0,C 180,E1 -14011.558,E2 -14011.558} C_VEL
LIN {X 0,Y 343.885,Z 847.449,A -85,B 0,C 180,E1 -14012.623,E2 -14012.623} C_VEL
LIN {X 0,Y 343.351,Z 855.582,A -85,B 0,C 180,E1 -14013.862,E2 -14013.862} C_VEL
LIN {X 0,Y 342.782,Z 862.731,A -85,B 0,C 180,E1 -14015.146,E2 -14015.146} C_VEL
LIN {X 0,Y 342.267,Z 868.704,A -85,B 0,C 180,E1 -14016.396,E2 -14016.396} C_VEL
LIN {X 0,Y 341.846,Z 874.008,A -85,B 0,C 180,E1 -14017.695,E2 -14017.695} C_VEL
LIN {X 0,Y 341.396,Z 880.015,A -85,B 0,C 180,E1 -14019.515,E2 -14019.515} C_VEL
LIN {X 0,Y 341.194,Z 883.416,A -85,B 0,C 180,E1 -14020.757,E2 -14020.757} C_VEL
LIN {X 0,Y 340.952,Z 887.417,A -85,B 0,C 180,E1 -14022.609,E2 -14022.609} C_VEL
LIN {X 0,Y 340.769,Z 890.259,A -85,B 0,C 180,E1 -14024.448,E2 -14024.448} C_VEL
LIN {X 0,Y 340.82,Z 892.41,A -85,B 0,C 180,E1 -14026.889,E2 -14026.889} C_VEL
LIN {X 0,Y 340.937,Z 892.808,A -85,B 0,C 180,E1 -14028.104,E2 -14028.104} C_VEL
LIN {X 0,Y 341.133,Z 892.748,A -85,B 0,C 180,E1 -14029.314,E2 -14029.314} C_VEL
LIN {X 0,Y 341.668,Z 891.332,A -85,B 0,C 180,E1 -14031.721,E2 -14031.721} C_VEL
LIN {X 0,Y 341.979,Z 889.938,A -85,B 0,C 180,E1 -14032.917,E2 -14032.917} C_VEL
LIN {X 0,Y 342.873,Z 885.817,A -85,B 0,C 180,E1 -14035.297,E2 -14035.297} C_VEL
LIN {X 0,Y 343.643,Z 881.42,A -85,B 0,C 180,E1 -14037.069,E2 -14037.069} C_VEL
LIN {X 0,Y 344.473,Z 876.355,A -85,B 0,C 180,E1 -14038.67,E2 -14038.67} C_VEL
LIN {X 0,Y 345.386,Z 871.216,A -85,B 0,C 180,E1 -14040,E2 -14040} C_VEL
LIN {X 0,Y 346.388,Z 864.437,A -85,B 0,C 180,E1 -14041.453,E2 -14041.453} C_VEL
LIN {X 0,Y 347.51,Z 856.18,A -85,B 0,C 180,E1 -14042.898,E2 -14042.898} C_VEL
LIN {X 0,Y 348.48,Z 848.309,A -85,B 0,C 180,E1 -14044.048,E2 -14044.048} C_VEL
LIN {X 0,Y 349.379,Z 840.176,A -85,B 0,C 180,E1 -14045.049,E2 -14045.049} C_VEL
LIN {X 0,Y 350.271,Z 830.335,A -85,B 0,C 180,E1 -14046.047,E2 -14046.047} C_VEL
LIN {X 0,Y 350.876,Z 821.88,A -85,B 0,C 180,E1 -14046.758,E2 -14046.758} C_VEL
LIN {X 0,Y 351.486,Z 811.204,A -85,B 0,C 180,E1 -14047.468,E2 -14047.468} C_VEL
LIN {X 0,Y 351.874,Z 800.678,A -85,B 0,C 180,E1 -14048.001,E2 -14048.001} C_VEL
LIN {X 0,Y 352.075,Z 788.113,A -85,B 0,C 180,E1 -14048.456,E2 -14048.456} C_VEL
LIN {X 0,Y 352.824,Z 764.498,A -85,B 0,C 180,E1 -14049.123,E2 -14049.123} C_VEL
LIN {X 0,Y 354.013,Z 735.573,A -85,B 0,C 180,E1 -14049.944,E2 -14049.944} C_VEL
LIN {X 0,Y 348.243,Z 723.848,A -85,B 0,C 180,E1 -14050.98,E2 -14050.98} C_VEL
LIN {X 0,Y 342.629,Z 713.931,A -85,B 0,C 180,E1 -14052.034,E2 -14052.034} C_VEL
LIN {X 0,Y 341.061,Z 711.072,A -85,B 0,C 180,E1 -14052.363,E2 -14052.363} C_VEL
LIN {X 0,Y 340.859,Z 710.154,A -85,B 0,C 180,E1 -14052.617,E2 -14052.617} C_VEL
LIN {X 0,Y 340.825,Z 710.032,A -85,B 0,C 180,E1 -14055.549,E2 -14055.549} C_VEL
LIN {X 0,Y 340.77,Z 710.038,A -85,B 0,C 180,E1 -14059.268,E2 -14059.268} C_VEL
LIN {X 0,Y 340.728,Z 710.042,A -85,B 0,C 180,E1 -14063.073,E2 -14063.073} C_VEL
LIN {X 0,Y 340.752,Z 710.04,A -85,B 0,C 180,E1 -14065.666,E2 -14065.666} C_VEL
LIN {X 0,Y 340.739,Z 710.042,A -85,B 0,C 180,E1 -14069.671,E2 -14069.671} C_VEL
LIN {X 0,Y 340.699,Z 710.046,A -85,B 0,C 180,E1 -14073.846,E2 -14073.846} C_VEL
LIN {X 0,Y 340.712,Z 710.042,A -85,B 0,C 180,E1 -14076.741,E2 -14076.741} C_VEL
LIN {X 0,Y 340.695,Z 710.047,A -85,B 0,C 180,E1 -14080.246,E2 -14080.246} C_VEL
LIN {X 0,Y 340.658,Z 710.052,A -85,B 0,C 180,E1 -14083.772,E2 -14083.772} C_VEL
LIN {X 0,Y 340.705,Z 710.047,A -85,B 0,C 180,E1 -14087.954,E2 -14087.954} C_VEL
LIN {X 0,Y 340.738,Z 710.044,A -85,B 0,C 180,E1 -14091.771,E2 -14091.771} C_VEL
LIN {X 0,Y 340.763,Z 710.242,A -85,B 0,C 180,E1 -14093.361,E2 -14093.361} C_VEL
LIN {X 0,Y 344.142,Z 724.192,A -85,B 0,C 180,E1 -14096.536,E2 -14096.536} C_VEL
LIN {X 0,Y 347.018,Z 737.009,A -85,B 0,C 180,E1 -14099.283,E2 -14099.283} C_VEL
LIN {X 0,Y 347.428,Z 740.12,A -85,B 0,C 180,E1 -14099.918,E2 -14099.918} C_VEL
LIN {X 0,Y 345.75,Z 755.462,A -85,B 0,C 180,E1 -14102.782,E2 -14102.782} C_VEL
LIN {X 0,Y 344.753,Z 766.447,A -85,B 0,C 180,E1 -14104.76,E2 -14104.76} C_VEL
LIN {X 0,Y 347.98,Z 790.328,A -85,B 0,C 180,E1 -14105.952,E2 -14105.952} C_VEL
LIN {X 0,Y 349.299,Z 803.125,A -85,B 0,C 180,E1 -14106.504,E2 -14106.504} C_VEL
LIN {X 0,Y 350.988,Z 830.49,A -85,B 0,C 180,E1 -14107.54,E2 -14107.54} C_VEL
LIN {X 0,Y 348.958,Z 882.528,A -85,B 0,C 180,E1 -14108.975,E2 -14108.975} C_VEL
LIN {X 0,Y 348.335,Z 893.039,A -85,B 0,C 180,E1 -14109.4,E2 -14109.4} C_VEL
LIN {X 0,Y 347.576,Z 902.369,A -85,B 0,C 180,E1 -14109.893,E2 -14109.893} C_VEL
LIN {X 0,Y 346.655,Z 911.091,A -85,B 0,C 180,E1 -14110.455,E2 -14110.455} C_VEL
LIN {X 0,Y 344.9,Z 926.909,A -85,B 0,C 180,E1 -14111.74,E2 -14111.74} C_VEL
LIN {X 0,Y 343.792,Z 937.025,A -85,B 0,C 180,E1 -14112.756,E2 -14112.756} C_VEL
LIN {X 0,Y 342.661,Z 946.502,A -85,B 0,C 180,E1 -14113.924,E2 -14113.924} C_VEL
LIN {X 0,Y 341.57,Z 956.281,A -85,B 0,C 180,E1 -14115.404,E2 -14115.404} C_VEL
LIN {X 0,Y 341.024,Z 962.781,A -85,B 0,C 180,E1 -14116.593,E2 -14116.593} C_VEL
LIN {X 0,Y 340.283,Z 970.962,A -85,B 0,C 180,E1 -14118.381,E2 -14118.381} C_VEL
LIN {X 0,Y 339.969,Z 976.531,A -85,B 0,C 180,E1 -14119.878,E2 -14119.878} C_VEL
LIN {X 0,Y 339.791,Z 981.99,A -85,B 0,C 180,E1 -14121.674,E2 -14121.674} C_VEL
LIN {X 0,Y 339.818,Z 985.421,A -85,B 0,C 180,E1 -14123.082,E2 -14123.082} C_VEL
LIN {X 0,Y 340.003,Z 989.41,A -85,B 0,C 180,E1 -14125.256,E2 -14125.256} C_VEL
LIN {X 0,Y 340.107,Z 990.964,A -85,B 0,C 180,E1 -14126.444,E2 -14126.444} C_VEL
LIN {X 0,Y 340.165,Z 992.035,A -85,B 0,C 180,E1 -14127.63,E2 -14127.63} C_VEL
LIN {X 0,Y 340.244,Z 992.693,A -85,B 0,C 180,E1 -14128.815,E2 -14128.815} C_VEL
LIN {X 0,Y 340.314,Z 992.94,A -85,B 0,C 180,E1 -14129.998,E2 -14129.998} C_VEL
LIN {X 0,Y 340.235,Z 992.753,A -85,B 0,C 180,E1 -14131.182,E2 -14131.182} C_VEL
LIN {X 0,Y 340.151,Z 992.111,A -85,B 0,C 180,E1 -14132.367,E2 -14132.367} C_VEL
LIN {X 0,Y 340.103,Z 991.061,A -85,B 0,C 180,E1 -14133.552,E2 -14133.552} C_VEL
LIN {X 0,Y 339.998,Z 989.587,A -85,B 0,C 180,E1 -14134.741,E2 -14134.741} C_VEL
LIN {X 0,Y 339.839,Z 985.67,A -85,B 0,C 180,E1 -14136.946,E2 -14136.946} C_VEL
LIN {X 0,Y 339.765,Z 980.758,A -85,B 0,C 180,E1 -14138.923,E2 -14138.923} C_VEL
LIN {X 0,Y 340.073,Z 974.011,A -85,B 0,C 180,E1 -14141.019,E2 -14141.019} C_VEL
LIN {X 0,Y 340.655,Z 966.734,A -85,B 0,C 180,E1 -14142.812,E2 -14142.812} C_VEL
LIN {X 0,Y 341.492,Z 959.38,A -85,B 0,C 180,E1 -14144.296,E2 -14144.296} C_VEL
LIN {X 0,Y 342.597,Z 949.523,A -85,B 0,C 180,E1 -14145.923,E2 -14145.923} C_VEL
LIN {X 0,Y 343.788,Z 939.69,A -85,B 0,C 180,E1 -14147.241,E2 -14147.241} C_VEL
LIN {X 0,Y 345.159,Z 929.016,A -85,B 0,C 180,E1 -14148.395,E2 -14148.395} C_VEL
LIN {X 0,Y 346.519,Z 917.267,A -85,B 0,C 180,E1 -14149.395,E2 -14149.395} C_VEL
LIN {X 0,Y 347.687,Z 905.135,A -85,B 0,C 180,E1 -14150.173,E2 -14150.173} C_VEL
LIN {X 0,Y 348.684,Z 892.066,A -85,B 0,C 180,E1 -14150.768,E2 -14150.768} C_VEL
LIN {X 0,Y 349.166,Z 878.146,A -85,B 0,C 180,E1 -14151.162,E2 -14151.162} C_VEL
LIN {X 0,Y 350.052,Z 828.193,A -85,B 0,C 180,E1 -14152.219,E2 -14152.219} C_VEL
LIN {X 0,Y 346.865,Z 795.587,A -85,B 0,C 180,E1 -14153.186,E2 -14153.186} C_VEL
LIN {X 0,Y 344.16,Z 774.307,A -85,B 0,C 180,E1 -14153.905,E2 -14153.905} C_VEL
LIN {X 0,Y 345.908,Z 756.457,A -85,B 0,C 180,E1 -14157.201,E2 -14157.201} C_VEL
LIN {X 0,Y 347.69,Z 741.199,A -85,B 0,C 180,E1 -14160.099,E2 -14160.099} C_VEL
LIN {X 0,Y 346.543,Z 734.232,A -85,B 0,C 180,E1 -14161.595,E2 -14161.595} C_VEL
LIN {X 0,Y 343.485,Z 720.649,A -85,B 0,C 180,E1 -14164.703,E2 -14164.703} C_VEL
LIN {X 0,Y 340.751,Z 710.146,A -85,B 0,C 180,E1 -14167.335,E2 -14167.335} C_VEL
LIN {X 0,Y 340.678,Z 710.049,A -85,B 0,C 180,E1 -14171.308,E2 -14171.308} C_VEL
LIN {X 0,Y 340.676,Z 710.051,A -85,B 0,C 180,E1 -14174.537,E2 -14174.537} C_VEL
LIN {X 0,Y 340.69,Z 710.048,A -85,B 0,C 180,E1 -14177.953,E2 -14177.953} C_VEL
LIN {X 0,Y 340.726,Z 710.042,A -85,B 0,C 180,E1 -14181.772,E2 -14181.772} C_VEL
LIN {X 0,Y 340.713,Z 710.034,A -85,B 0,C 180,E1 -14185.594,E2 -14185.594} C_VEL
LIN {X 0,Y 340.694,Z 710.044,A -85,B 0,C 180,E1 -14188.955,E2 -14188.955} C_VEL
LIN {X 0,Y 340.769,Z 710.033,A -85,B 0,C 180,E1 -14192.473,E2 -14192.473} C_VEL
LIN {X 0,Y 340.745,Z 710.037,A -85,B 0,C 180,E1 -14195.638,E2 -14195.638} C_VEL
LIN {X 0,Y 340.736,Z 710.036,A -85,B 0,C 180,E1 -14199.474,E2 -14199.474} C_VEL
LIN {X 0,Y 340.847,Z 710.021,A -85,B 0,C 180,E1 -14201.984,E2 -14201.984} C_VEL
LIN {X 0,Y 340.857,Z 710.023,A -85,B 0,C 180,E1 -14205.705,E2 -14205.705} C_VEL
LIN {X 0,Y 340.859,Z 710.025,A -85,B 0,C 180,E1 -14209.306,E2 -14209.306} C_VEL
LIN {X 0,Y 341.046,Z 710.001,A -85,B 0,C 180,E1 -14212.898,E2 -14212.898} C_VEL
LIN {X 0,Y 341.159,Z 709.986,A -85,B 0,C 180,E1 -14217.639,E2 -14217.639} C_VEL
LIN {X 0,Y 341.284,Z 709.966,A -85,B 0,C 180,E1 -14220,E2 -14220} C_VEL
LIN {X 0,Y 341.158,Z 709.99,A -85,B 0,C 180,E1 -14222.362,E2 -14222.362} C_VEL
LIN {X 0,Y 341.063,Z 709.999,A -85,B 0,C 180,E1 -14227.102,E2 -14227.102} C_VEL
LIN {X 0,Y 340.859,Z 710.029,A -85,B 0,C 180,E1 -14230.694,E2 -14230.694} C_VEL
LIN {X 0,Y 340.852,Z 710.027,A -85,B 0,C 180,E1 -14234.326,E2 -14234.326} C_VEL
LIN {X 0,Y 340.826,Z 710.03,A -85,B 0,C 180,E1 -14238.467,E2 -14238.467} C_VEL
LIN {X 0,Y 340.707,Z 710.04,A -85,B 0,C 180,E1 -14241.843,E2 -14241.843} C_VEL
LIN {X 0,Y 340.761,Z 710.04,A -85,B 0,C 180,E1 -14245.666,E2 -14245.666} C_VEL
LIN {X 0,Y 340.718,Z 710.03,A -85,B 0,C 180,E1 -14248.322,E2 -14248.322} C_VEL
LIN {X 0,Y 340.688,Z 710.052,A -85,B 0,C 180,E1 -14251.046,E2 -14251.046} C_VEL
LIN {X 0,Y 340.71,Z 710.04,A -85,B 0,C 180,E1 -14255.28,E2 -14255.28} C_VEL
LIN {X 0,Y 340.704,Z 710.04,A -85,B 0,C 180,E1 -14258.388,E2 -14258.388} C_VEL
LIN {X 0,Y 340.726,Z 710.276,A -85,B 0,C 180,E1 -14261.231,E2 -14261.231} C_VEL
LIN {X 0,Y 341.008,Z 711.469,A -85,B 0,C 180,E1 -14261.436,E2 -14261.436} C_VEL
LIN {X 0,Y 348.222,Z 726.617,A -85,B 0,C 180,E1 -14262.394,E2 -14262.394} C_VEL
LIN {X 0,Y 351.751,Z 735.22,A -85,B 0,C 180,E1 -14262.864,E2 -14262.864} C_VEL
LIN {X 0,Y 350.897,Z 786.587,A -85,B 0,C 180,E1 -14263.971,E2 -14263.971} C_VEL
LIN {X 0,Y 350.824,Z 800.034,A -85,B 0,C 180,E1 -14264.374,E2 -14264.374} C_VEL
LIN {X 0,Y 350.513,Z 812.578,A -85,B 0,C 180,E1 -14264.984,E2 -14264.984} C_VEL
LIN {X 0,Y 349.888,Z 825.042,A -85,B 0,C 180,E1 -14265.828,E2 -14265.828} C_VEL
LIN {X 0,Y 349.057,Z 836.02,A -85,B 0,C 180,E1 -14266.801,E2 -14266.801} C_VEL
LIN {X 0,Y 348.043,Z 846.799,A -85,B 0,C 180,E1 -14268.021,E2 -14268.021} C_VEL
LIN {X 0,Y 346.929,Z 856.618,A -85,B 0,C 180,E1 -14269.402,E2 -14269.402} C_VEL
LIN {X 0,Y 345.801,Z 865.51,A -85,B 0,C 180,E1 -14270.95,E2 -14270.95} C_VEL
LIN {X 0,Y 344.562,Z 874.036,A -85,B 0,C 180,E1 -14272.821,E2 -14272.821} C_VEL
LIN {X 0,Y 343.772,Z 879.674,A -85,B 0,C 180,E1 -14274.366,E2 -14274.366} C_VEL
LIN {X 0,Y 342.778,Z 885.556,A -85,B 0,C 180,E1 -14276.389,E2 -14276.389} C_VEL
LIN {X 0,Y 342.089,Z 889.894,A -85,B 0,C 180,E1 -14278.409,E2 -14278.409} C_VEL
LIN {X 0,Y 341.574,Z 892.87,A -85,B 0,C 180,E1 -14280.411,E2 -14280.411} C_VEL
LIN {X 0,Y 341.276,Z 894.599,A -85,B 0,C 180,E1 -14282.316,E2 -14282.316} C_VEL
LIN {X 0,Y 341.043,Z 895.32,A -85,B 0,C 180,E1 -14284.36,E2 -14284.36} C_VEL
LIN {X 0,Y 340.964,Z 895.195,A -85,B 0,C 180,E1 -14285.656,E2 -14285.656} C_VEL
LIN {X 0,Y 341.106,Z 893.718,A -85,B 0,C 180,E1 -14287.998,E2 -14287.998} C_VEL
LIN {X 0,Y 341.474,Z 890.98,A -85,B 0,C 180,E1 -14290.15,E2 -14290.15} C_VEL
LIN {X 0,Y 341.931,Z 887.399,A -85,B 0,C 180,E1 -14292.045,E2 -14292.045} C_VEL
LIN {X 0,Y 342.567,Z 882.637,A -85,B 0,C 180,E1 -14293.924,E2 -14293.924} C_VEL
LIN {X 0,Y 343.332,Z 876.547,A -85,B 0,C 180,E1 -14295.782,E2 -14295.782} C_VEL
LIN {X 0,Y 344.271,Z 868.649,A -85,B 0,C 180,E1 -14297.684,E2 -14297.684} C_VEL
LIN {X 0,Y 345.147,Z 861.092,A -85,B 0,C 180,E1 -14299.156,E2 -14299.156} C_VEL
LIN {X 0,Y 346.134,Z 851.722,A -85,B 0,C 180,E1 -14300.654,E2 -14300.654} C_VEL
LIN {X 0,Y 347.111,Z 841.266,A -85,B 0,C 180,E1 -14301.991,E2 -14301.991} C_VEL
LIN {X 0,Y 348.089,Z 829.468,A -85,B 0,C 180,E1 -14303.189,E2 -14303.189} C_VEL
LIN {X 0,Y 348.769,Z 817.252,A -85,B 0,C 180,E1 -14304.147,E2 -14304.147} C_VEL
LIN {X 0,Y 349.209,Z 804.579,A -85,B 0,C 180,E1 -14304.878,E2 -14304.878} C_VEL
LIN {X 0,Y 349.415,Z 791.613,A -85,B 0,C 180,E1 -14305.387,E2 -14305.387} C_VEL
LIN {X 0,Y 349.924,Z 746.147,A -85,B 0,C 180,E1 -14306.382,E2 -14306.382} C_VEL
LIN {X 0,Y 350.127,Z 732.537,A -85,B 0,C 180,E1 -14306.671,E2 -14306.671} C_VEL
LIN {X 0,Y 341.323,Z 710.942,A -85,B 0,C 180,E1 -14307.752,E2 -14307.752} C_VEL
LIN {X 0,Y 341.121,Z 710.054,A -85,B 0,C 180,E1 -14308.009,E2 -14308.009} C_VEL
LIN {X 0,Y 341.091,Z 709.998,A -85,B 0,C 180,E1 -14311.182,E2 -14311.182} C_VEL
LIN {X 0,Y 341.12,Z 709.992,A -85,B 0,C 180,E1 -14312.363,E2 -14312.363} C_VEL
LIN {X 0,Y 341.015,Z 710.01,A -85,B 0,C 180,E1 -14315.916,E2 -14315.916} C_VEL
LIN {X 0,Y 340.968,Z 710.011,A -85,B 0,C 180,E1 -14318.358,E2 -14318.358} C_VEL
LIN {X 0,Y 340.849,Z 710.024,A -85,B 0,C 180,E1 -14321.901,E2 -14321.901} C_VEL
LIN {X 0,Y 340.822,Z 710.024,A -85,B 0,C 180,E1 -14325.551,E2 -14325.551} C_VEL
LIN {X 0,Y 340.723,Z 710.03,A -85,B 0,C 180,E1 -14329.272,E2 -14329.272} C_VEL
LIN {X 0,Y 340.706,Z 710.047,A -85,B 0,C 180,E1 -14333.076,E2 -14333.076} C_VEL
LIN {X 0,Y 340.716,Z 710.025,A -85,B 0,C 180,E1 -14336.989,E2 -14336.989} C_VEL
LIN {X 0,Y 340.723,Z 710.041,A -85,B 0,C 180,E1 -14339.965,E2 -14339.965} C_VEL
LIN {X 0,Y 340.678,Z 710.038,A -85,B 0,C 180,E1 -14342.604,E2 -14342.604} C_VEL
LIN {X 0,Y 339.996,Z 710.112,A -85,B 0,C 180,E1 -14343.591,E2 -14343.591} C_VEL
LIN {X 0,Y 337.175,Z 710.466,A -85,B 0,C 180,E1 -14345.198,E2 -14345.198} C_VEL
LIN {X 0,Y 334.783,Z 710.772,A -85,B 0,C 180,E1 -14346.499,E2 -14346.499} C_VEL
LIN {X 0,Y 333.734,Z 710.906,A -85,B 0,C 180,E1 -14347.504,E2 -14347.504} C_VEL
LIN {X 0,Y 333.635,Z 710.918,A -85,B 0,C 180,E1 -14347.845,E2 -14347.845} C_VEL
LIN {X 0,Y 333.603,Z 710.928,A -85,B 0,C 180,E1 -14350.776,E2 -14350.776} C_VEL
LIN {X 0,Y 333.589,Z 710.931,A -85,B 0,C 180,E1 -14354.249,E2 -14354.249} C_VEL
LIN {X 0,Y 333.642,Z 710.927,A -85,B 0,C 180,E1 -14357.618,E2 -14357.618} C_VEL
LIN {X 0,Y 333.622,Z 710.928,A -85,B 0,C 180,E1 -14361.211,E2 -14361.211} C_VEL
LIN {X 0,Y 333.753,Z 711.121,A -85,B 0,C 180,E1 -14365.055,E2 -14365.055} C_VEL
LIN {X 0,Y 333.944,Z 712.021,A -85,B 0,C 180,E1 -14365.233,E2 -14365.233} C_VEL
LIN {X 0,Y 341.089,Z 732.209,A -85,B 0,C 180,E1 -14366.165,E2 -14366.165} C_VEL
LIN {X 0,Y 339.863,Z 787.743,A -85,B 0,C 180,E1 -14367.613,E2 -14367.613} C_VEL
LIN {X 0,Y 339.628,Z 799.755,A -85,B 0,C 180,E1 -14368.106,E2 -14368.106} C_VEL
LIN {X 0,Y 339.299,Z 810.121,A -85,B 0,C 180,E1 -14368.689,E2 -14368.689} C_VEL
LIN {X 0,Y 338.774,Z 820.675,A -85,B 0,C 180,E1 -14369.451,E2 -14369.451} C_VEL
LIN {X 0,Y 338.187,Z 830.423,A -85,B 0,C 180,E1 -14370.325,E2 -14370.325} C_VEL
LIN {X 0,Y 337.552,Z 840.131,A -85,B 0,C 180,E1 -14371.388,E2 -14371.388} C_VEL
LIN {X 0,Y 336.899,Z 848.716,A -85,B 0,C 180,E1 -14372.513,E2 -14372.513} C_VEL
LIN {X 0,Y 336.385,Z 856.047,A -85,B 0,C 180,E1 -14373.642,E2 -14373.642} C_VEL
LIN {X 0,Y 335.816,Z 863.168,A -85,B 0,C 180,E1 -14374.925,E2 -14374.925} C_VEL
LIN {X 0,Y 335.125,Z 870.538,A -85,B 0,C 180,E1 -14376.518,E2 -14376.518} C_VEL
LIN {X 0,Y 334.687,Z 876.626,A -85,B 0,C 180,E1 -14378.116,E2 -14378.116} C_VEL
LIN {X 0,Y 334.321,Z 881.613,A -85,B 0,C 180,E1 -14379.704,E2 -14379.704} C_VEL
LIN {X 0,Y 334.049,Z 885.516,A -85,B 0,C 180,E1 -14381.222,E2 -14381.222} C_VEL
LIN {X 0,Y 333.873,Z 888.833,A -85,B 0,C 180,E1 -14382.86,E2 -14382.86} C_VEL
LIN {X 0,Y 333.767,Z 890.766,A -85,B 0,C 180,E1 -14384.113,E2 -14384.113} C_VEL
LIN {X 0,Y 333.795,Z 893.263,A -85,B 0,C 180,E1 -14386.608,E2 -14386.608} C_VEL
LIN {X 0,Y 333.908,Z 893.83,A -85,B 0,C 180,E1 -14387.849,E2 -14387.849} C_VEL
LIN {X 0,Y 334.107,Z 893.942,A -85,B 0,C 180,E1 -14389.087,E2 -14389.087} C_VEL
LIN {X 0,Y 334.654,Z 892.825,A -85,B 0,C 180,E1 -14391.546,E2 -14391.546} C_VEL
LIN {X 0,Y 335.386,Z 889.904,A -85,B 0,C 180,E1 -14393.986,E2 -14393.986} C_VEL
LIN {X 0,Y 336.123,Z 886.517,A -85,B 0,C 180,E1 -14395.803,E2 -14395.803} C_VEL
LIN {X 0,Y 336.698,Z 883.721,A -85,B 0,C 180,E1 -14397.009,E2 -14397.009} C_VEL
LIN {X 0,Y 337.642,Z 878.342,A -85,B 0,C 180,E1 -14398.807,E2 -14398.807} C_VEL
LIN {X 0,Y 338.905,Z 871.462,A -85,B 0,C 180,E1 -14400.594,E2 -14400.594} C_VEL
LIN {X 0,Y 339.985,Z 864.551,A -85,B 0,C 180,E1 -14402.073,E2 -14402.073} C_VEL
LIN {X 0,Y 340.975,Z 857.99,A -85,B 0,C 180,E1 -14403.249,E2 -14403.249} C_VEL
LIN {X 0,Y 342.013,Z 850.245,A -85,B 0,C 180,E1 -14404.419,E2 -14404.419} C_VEL
LIN {X 0,Y 343.082,Z 840.924,A -85,B 0,C 180,E1 -14405.584,E2 -14405.584} C_VEL
LIN {X 0,Y 343.889,Z 832.583,A -85,B 0,C 180,E1 -14406.454,E2 -14406.454} C_VEL
LIN {X 0,Y 344.658,Z 822.369,A -85,B 0,C 180,E1 -14407.322,E2 -14407.322} C_VEL
LIN {X 0,Y 345.307,Z 811.608,A -85,B 0,C 180,E1 -14408.043,E2 -14408.043} C_VEL
LIN {X 0,Y 345.706,Z 801.803,A -85,B 0,C 180,E1 -14408.549,E2 -14408.549} C_VEL
LIN {X 0,Y 345.972,Z 788.009,A -85,B 0,C 180,E1 -14409.058,E2 -14409.058} C_VEL
LIN {X 0,Y 347.179,Z 755.976,A -85,B 0,C 180,E1 -14409.99,E2 -14409.99} C_VEL
LIN {X 0,Y 348.052,Z 737.898,A -85,B 0,C 180,E1 -14410.511,E2 -14410.511} C_VEL
LIN {X 0,Y 341.809,Z 725.354,A -85,B 0,C 180,E1 -14411.709,E2 -14411.709} C_VEL
LIN {X 0,Y 337.307,Z 717.758,A -85,B 0,C 180,E1 -14412.585,E2 -14412.585} C_VEL
LIN {X 0,Y 335.694,Z 714.918,A -85,B 0,C 180,E1 -14412.922,E2 -14412.922} C_VEL
LIN {X 0,Y 334.073,Z 712.088,A -85,B 0,C 180,E1 -14413.284,E2 -14413.284} C_VEL
LIN {X 0,Y 333.841,Z 711.111,A -85,B 0,C 180,E1 -14413.518,E2 -14413.518} C_VEL
LIN {X 0,Y 333.781,Z 710.91,A -85,B 0,C 180,E1 -14415.886,E2 -14415.886} C_VEL
LIN {X 0,Y 333.725,Z 710.916,A -85,B 0,C 180,E1 -14419.691,E2 -14419.691} C_VEL
LIN {X 0,Y 333.675,Z 710.919,A -85,B 0,C 180,E1 -14423.59,E2 -14423.59} C_VEL
LIN {X 0,Y 333.683,Z 710.922,A -85,B 0,C 180,E1 -14426.251,E2 -14426.251} C_VEL
LIN {X 0,Y 333.667,Z 710.921,A -85,B 0,C 180,E1 -14430.365,E2 -14430.365} C_VEL
LIN {X 0,Y 333.644,Z 710.926,A -85,B 0,C 180,E1 -14433.208,E2 -14433.208} C_VEL
LIN {X 0,Y 333.683,Z 710.92,A -85,B 0,C 180,E1 -14436.138,E2 -14436.138} C_VEL
LIN {X 0,Y 333.654,Z 710.922,A -85,B 0,C 180,E1 -14439.191,E2 -14439.191} C_VEL
LIN {X 0,Y 333.639,Z 710.926,A -85,B 0,C 180,E1 -14442.499,E2 -14442.499} C_VEL
LIN {X 0,Y 333.603,Z 710.932,A -85,B 0,C 180,E1 -14445.954,E2 -14445.954} C_VEL
LIN {X 0,Y 333.653,Z 710.923,A -85,B 0,C 180,E1 -14449.314,E2 -14449.314} C_VEL
LIN {X 0,Y 333.731,Z 711.129,A -85,B 0,C 180,E1 -14452.925,E2 -14452.925} C_VEL
LIN {X 0,Y 337.124,Z 725.099,A -85,B 0,C 180,E1 -14456.19,E2 -14456.19} C_VEL
LIN {X 0,Y 340.22,Z 739.058,A -85,B 0,C 180,E1 -14459.25,E2 -14459.25} C_VEL
LIN {X 0,Y 340.465,Z 742.713,A -85,B 0,C 180,E1 -14459.994,E2 -14459.994} C_VEL
LIN {X 0,Y 338.176,Z 763.366,A -85,B 0,C 180,E1 -14463.873,E2 -14463.873} C_VEL
LIN {X 0,Y 341.613,Z 788.354,A -85,B 0,C 180,E1 -14465.201,E2 -14465.201} C_VEL
LIN {X 0,Y 343.238,Z 804.692,A -85,B 0,C 180,E1 -14465.944,E2 -14465.944} C_VEL
LIN {X 0,Y 344.795,Z 831.004,A -85,B 0,C 180,E1 -14466.981,E2 -14466.981} C_VEL
LIN {X 0,Y 342.665,Z 881.161,A -85,B 0,C 180,E1 -14468.412,E2 -14468.412} C_VEL
LIN {X 0,Y 341.949,Z 891.565,A -85,B 0,C 180,E1 -14468.839,E2 -14468.839} C_VEL
LIN {X 0,Y 341.07,Z 902.086,A -85,B 0,C 180,E1 -14469.414,E2 -14469.414} C_VEL
LIN {X 0,Y 340.009,Z 911.534,A -85,B 0,C 180,E1 -14470.057,E2 -14470.057} C_VEL
LIN {X 0,Y 338.739,Z 921.884,A -85,B 0,C 180,E1 -14470.925,E2 -14470.925} C_VEL
LIN {X 0,Y 336.947,Z 935.746,A -85,B 0,C 180,E1 -14472.394,E2 -14472.394} C_VEL
LIN {X 0,Y 335.661,Z 946.359,A -85,B 0,C 180,E1 -14473.735,E2 -14473.735} C_VEL
LIN {X 0,Y 334.743,Z 954.32,A -85,B 0,C 180,E1 -14474.968,E2 -14474.968} C_VEL
LIN {X 0,Y 334.095,Z 961.617,A -85,B 0,C 180,E1 -14476.309,E2 -14476.309} C_VEL
LIN {X 0,Y 333.278,Z 969.825,A -85,B 0,C 180,E1 -14478.133,E2 -14478.133} C_VEL
LIN {X 0,Y 332.905,Z 975.416,A -85,B 0,C 180,E1 -14479.661,E2 -14479.661} C_VEL
LIN {X 0,Y 332.743,Z 980.905,A -85,B 0,C 180,E1 -14481.496,E2 -14481.496} C_VEL
LIN {X 0,Y 332.753,Z 984.622,A -85,B 0,C 180,E1 -14483.063,E2 -14483.063} C_VEL
LIN {X 0,Y 332.946,Z 988.36,A -85,B 0,C 180,E1 -14485.155,E2 -14485.155} C_VEL
LIN {X 0,Y 333.062,Z 989.927,A -85,B 0,C 180,E1 -14486.369,E2 -14486.369} C_VEL
LIN {X 0,Y 333.123,Z 991.009,A -85,B 0,C 180,E1 -14487.58,E2 -14487.58} C_VEL
LIN {X 0,Y 333.209,Z 991.673,A -85,B 0,C 180,E1 -14488.79,E2 -14488.79} C_VEL
LIN {X 0,Y 333.286,Z 991.927,A -85,B 0,C 180,E1 -14489.998,E2 -14489.998} C_VEL
LIN {X 0,Y 333.198,Z 991.746,A -85,B 0,C 180,E1 -14491.207,E2 -14491.207} C_VEL
LIN {X 0,Y 333.107,Z 991.111,A -85,B 0,C 180,E1 -14492.417,E2 -14492.417} C_VEL
LIN {X 0,Y 333.058,Z 990.064,A -85,B 0,C 180,E1 -14493.628,E2 -14493.628} C_VEL
LIN {X 0,Y 332.941,Z 988.594,A -85,B 0,C 180,E1 -14494.842,E2 -14494.842} C_VEL
LIN {X 0,Y 332.768,Z 984.978,A -85,B 0,C 180,E1 -14496.959,E2 -14496.959} C_VEL
LIN {X 0,Y 332.71,Z 979.799,A -85,B 0,C 180,E1 -14499.114,E2 -14499.114} C_VEL
LIN {X 0,Y 333.061,Z 973.071,A -85,B 0,C 180,E1 -14501.254,E2 -14501.254} C_VEL
LIN {X 0,Y 333.657,Z 965.815,A -85,B 0,C 180,E1 -14503.085,E2 -14503.085} C_VEL
LIN {X 0,Y 334.418,Z 960.034,A -85,B 0,C 180,E1 -14504.294,E2 -14504.294} C_VEL
LIN {X 0,Y 335.274,Z 952.648,A -85,B 0,C 180,E1 -14505.625,E2 -14505.625} C_VEL
LIN {X 0,Y 336.298,Z 943.45,A -85,B 0,C 180,E1 -14507.01,E2 -14507.01} C_VEL
LIN {X 0,Y 337.877,Z 932.528,A -85,B 0,C 180,E1 -14508.335,E2 -14508.335} C_VEL
LIN {X 0,Y 339.134,Z 921.963,A -85,B 0,C 180,E1 -14509.362,E2 -14509.362} C_VEL
LIN {X 0,Y 340.544,Z 909.346,A -85,B 0,C 180,E1 -14510.3,E2 -14510.3} C_VEL
LIN {X 0,Y 341.738,Z 896.142,A -85,B 0,C 180,E1 -14511.013,E2 -14511.013} C_VEL
LIN {X 0,Y 342.438,Z 883.056,A -85,B 0,C 180,E1 -14511.48,E2 -14511.48} C_VEL
LIN {X 0,Y 343.521,Z 828.846,A -85,B 0,C 180,E1 -14512.665,E2 -14512.665} C_VEL
LIN {X 0,Y 340.276,Z 795.472,A -85,B 0,C 180,E1 -14513.684,E2 -14513.684} C_VEL
LIN {X 0,Y 337.411,Z 773.035,A -85,B 0,C 180,E1 -14514.48,E2 -14514.48} C_VEL
LIN {X 0,Y 339.195,Z 755.63,A -85,B 0,C 180,E1 -14517.785,E2 -14517.785} C_VEL
LIN {X 0,Y 340.738,Z 743.817,A -85,B 0,C 180,E1 -14520.075,E2 -14520.075} C_VEL
LIN {X 0,Y 340.662,Z 740.682,A -85,B 0,C 180,E1 -14520.724,E2 -14520.724} C_VEL
LIN {X 0,Y 337.905,Z 727.659,A -85,B 0,C 180,E1 -14523.7,E2 -14523.7} C_VEL
LIN {X 0,Y 334.957,Z 715.802,A -85,B 0,C 180,E1 -14526.61,E2 -14526.61} C_VEL
LIN {X 0,Y 333.697,Z 710.997,A -85,B 0,C 180,E1 -14527.929,E2 -14527.929} C_VEL
LIN {X 0,Y 333.639,Z 710.922,A -85,B 0,C 180,E1 -14530.766,E2 -14530.766} C_VEL
LIN {X 0,Y 333.619,Z 710.928,A -85,B 0,C 180,E1 -14534.255,E2 -14534.255} C_VEL
LIN {X 0,Y 333.633,Z 710.927,A -85,B 0,C 180,E1 -14537.617,E2 -14537.617} C_VEL
LIN {X 0,Y 333.645,Z 710.918,A -85,B 0,C 180,E1 -14541.2,E2 -14541.2} C_VEL
LIN {X 0,Y 333.668,Z 710.91,A -85,B 0,C 180,E1 -14543.86,E2 -14543.86} C_VEL
LIN {X 0,Y 333.636,Z 710.928,A -85,B 0,C 180,E1 -14547.411,E2 -14547.411} C_VEL
LIN {X 0,Y 333.701,Z 710.918,A -85,B 0,C 180,E1 -14551.027,E2 -14551.027} C_VEL
LIN {X 0,Y 333.725,Z 710.914,A -85,B 0,C 180,E1 -14553.753,E2 -14553.753} C_VEL
LIN {X 0,Y 333.708,Z 710.912,A -85,B 0,C 180,E1 -14557.913,E2 -14557.913} C_VEL
LIN {X 0,Y 333.783,Z 710.905,A -85,B 0,C 180,E1 -14561.589,E2 -14561.589} C_VEL
LIN {X 0,Y 333.796,Z 710.904,A -85,B 0,C 180,E1 -14565.576,E2 -14565.576} C_VEL
LIN {X 0,Y 333.822,Z 710.901,A -85,B 0,C 180,E1 -14569.078,E2 -14569.078} C_VEL
LIN {X 0,Y 333.993,Z 710.88,A -85,B 0,C 180,E1 -14572.747,E2 -14572.747} C_VEL
LIN {X 0,Y 333.799,Z 710.898,A -85,B 0,C 180,E1 -14575.169,E2 -14575.169} C_VEL
LIN {X 0,Y 334.096,Z 710.866,A -85,B 0,C 180,E1 -14577.589,E2 -14577.589} C_VEL
LIN {X 0,Y 334.235,Z 710.843,A -85,B 0,C 180,E1 -14580,E2 -14580} C_VEL
LIN {X 0,Y 334.095,Z 710.87,A -85,B 0,C 180,E1 -14582.411,E2 -14582.411} C_VEL
LIN {X 0,Y 334.013,Z 710.876,A -85,B 0,C 180,E1 -14587.253,E2 -14587.253} C_VEL
LIN {X 0,Y 333.822,Z 710.903,A -85,B 0,C 180,E1 -14590.923,E2 -14590.923} C_VEL
LIN {X 0,Y 333.797,Z 710.908,A -85,B 0,C 180,E1 -14594.635,E2 -14594.635} C_VEL
LIN {X 0,Y 333.785,Z 710.906,A -85,B 0,C 180,E1 -14598.656,E2 -14598.656} C_VEL
LIN {X 0,Y 333.646,Z 710.916,A -85,B 0,C 180,E1 -14602.282,E2 -14602.282} C_VEL
LIN {X 0,Y 333.724,Z 710.917,A -85,B 0,C 180,E1 -14606.248,E2 -14606.248} C_VEL
LIN {X 0,Y 333.68,Z 710.907,A -85,B 0,C 180,E1 -14608.975,E2 -14608.975} C_VEL
LIN {X 0,Y 333.636,Z 710.915,A -85,B 0,C 180,E1 -14612.589,E2 -14612.589} C_VEL
LIN {X 0,Y 333.669,Z 710.914,A -85,B 0,C 180,E1 -14616.14,E2 -14616.14} C_VEL
LIN {X 0,Y 333.651,Z 710.928,A -85,B 0,C 180,E1 -14619.945,E2 -14619.945} C_VEL
LIN {X 0,Y 333.699,Z 711.219,A -85,B 0,C 180,E1 -14620.669,E2 -14620.669} C_VEL
LIN {X 0,Y 334.023,Z 712.479,A -85,B 0,C 180,E1 -14620.86,E2 -14620.86} C_VEL
LIN {X 0,Y 341.523,Z 727.828,A -85,B 0,C 180,E1 -14621.882,E2 -14621.882} C_VEL
LIN {X 0,Y 345.317,Z 736.832,A -85,B 0,C 180,E1 -14622.403,E2 -14622.403} C_VEL
LIN {X 0,Y 344.4,Z 786.709,A -85,B 0,C 180,E1 -14623.499,E2 -14623.499} C_VEL
LIN {X 0,Y 344.313,Z 800.871,A -85,B 0,C 180,E1 -14623.922,E2 -14623.922} C_VEL
LIN {X 0,Y 343.985,Z 813.73,A -85,B 0,C 180,E1 -14624.562,E2 -14624.562} C_VEL
LIN {X 0,Y 343.36,Z 825.77,A -85,B 0,C 180,E1 -14625.39,E2 -14625.39} C_VEL
LIN {X 0,Y 342.486,Z 836.745,A -85,B 0,C 180,E1 -14626.372,E2 -14626.372} C_VEL
LIN {X 0,Y 341.403,Z 847.767,A -85,B 0,C 180,E1 -14627.638,E2 -14627.638} C_VEL
LIN {X 0,Y 340.109,Z 858.575,A -85,B 0,C 180,E1 -14629.197,E2 -14629.197} C_VEL
LIN {X 0,Y 338.931,Z 867.244,A -85,B 0,C 180,E1 -14630.772,E2 -14630.772} C_VEL
LIN {X 0,Y 337.755,Z 875.054,A -85,B 0,C 180,E1 -14632.534,E2 -14632.534} C_VEL
LIN {X 0,Y 336.7,Z 881.939,A -85,B 0,C 180,E1 -14634.495,E2 -14634.495} C_VEL
LIN {X 0,Y 335.803,Z 886.942,A -85,B 0,C 180,E1 -14636.319,E2 -14636.319} C_VEL
LIN {X 0,Y 335.111,Z 891.152,A -85,B 0,C 180,E1 -14638.381,E2 -14638.381} C_VEL
LIN {X 0,Y 334.713,Z 893.225,A -85,B 0,C 180,E1 -14639.742,E2 -14639.742} C_VEL
LIN {X 0,Y 334.286,Z 895.492,A -85,B 0,C 180,E1 -14642.008,E2 -14642.008} C_VEL
LIN {X 0,Y 334.068,Z 896.287,A -85,B 0,C 180,E1 -14643.784,E2 -14643.784} C_VEL
LIN {X 0,Y 333.97,Z 896.307,A -85,B 0,C 180,E1 -14645.112,E2 -14645.112} C_VEL
LIN {X 0,Y 333.95,Z 895.88,A -85,B 0,C 180,E1 -14646.433,E2 -14646.433} C_VEL
LIN {X 0,Y 334.067,Z 894.978,A -85,B 0,C 180,E1 -14647.769,E2 -14647.769} C_VEL
LIN {X 0,Y 334.266,Z 893.603,A -85,B 0,C 180,E1 -14649.06,E2 -14649.06} C_VEL
LIN {X 0,Y 334.622,Z 890.804,A -85,B 0,C 180,E1 -14650.932,E2 -14650.932} C_VEL
LIN {X 0,Y 335.197,Z 886.62,A -85,B 0,C 180,E1 -14652.932,E2 -14652.932} C_VEL
LIN {X 0,Y 335.93,Z 881.13,A -85,B 0,C 180,E1 -14654.915,E2 -14654.915} C_VEL
LIN {X 0,Y 336.735,Z 874.706,A -85,B 0,C 180,E1 -14656.73,E2 -14656.73} C_VEL
LIN {X 0,Y 337.655,Z 867.665,A -85,B 0,C 180,E1 -14658.334,E2 -14658.334} C_VEL
LIN {X 0,Y 338.558,Z 859.661,A -85,B 0,C 180,E1 -14659.839,E2 -14659.839} C_VEL
LIN {X 0,Y 339.651,Z 849.609,A -85,B 0,C 180,E1 -14661.374,E2 -14661.374} C_VEL
LIN {X 0,Y 340.667,Z 838.288,A -85,B 0,C 180,E1 -14662.752,E2 -14662.752} C_VEL
LIN {X 0,Y 341.539,Z 827.317,A -85,B 0,C 180,E1 -14663.8,E2 -14663.8} C_VEL
LIN {X 0,Y 342.199,Z 815.25,A -85,B 0,C 180,E1 -14664.699,E2 -14664.699} C_VEL
LIN {X 0,Y 342.598,Z 802.903,A -85,B 0,C 180,E1 -14665.374,E2 -14665.374} C_VEL
LIN {X 0,Y 342.736,Z 790.508,A -85,B 0,C 180,E1 -14665.823,E2 -14665.823} C_VEL
LIN {X 0,Y 343.552,Z 734.316,A -85,B 0,C 180,E1 -14667.052,E2 -14667.052} C_VEL
LIN {X 0,Y 334.238,Z 711.761,A -85,B 0,C 180,E1 -14668.234,E2 -14668.234} C_VEL
LIN {X 0,Y 334.056,Z 710.935,A -85,B 0,C 180,E1 -14668.491,E2 -14668.491} C_VEL
LIN {X 0,Y 334.061,Z 710.872,A -85,B 0,C 180,E1 -14672.413,E2 -14672.413} C_VEL
LIN {X 0,Y 333.989,Z 710.886,A -85,B 0,C 180,E1 -14676.041,E2 -14676.041} C_VEL
LIN {X 0,Y 333.917,Z 710.891,A -85,B 0,C 180,E1 -14678.474,E2 -14678.474} C_VEL
LIN {X 0,Y 333.792,Z 710.904,A -85,B 0,C 180,E1 -14682.156,E2 -14682.156} C_VEL
LIN {X 0,Y 333.814,Z 710.894,A -85,B 0,C 180,E1 -14684.636,E2 -14684.636} C_VEL
LIN {X 0,Y 333.712,Z 710.91,A -85,B 0,C 180,E1 -14688.61,E2 -14688.61} C_VEL
LIN {X 0,Y 333.655,Z 710.92,A -85,B 0,C 180,E1 -14692.283,E2 -14692.283} C_VEL
LIN {X 0,Y 333.665,Z 710.911,A -85,B 0,C 180,E1 -14695.08,E2 -14695.08} C_VEL
LIN {X 0,Y 333.634,Z 710.92,A -85,B 0,C 180,E1 -14698.981,E2 -14698.981} C_VEL
LIN {X 0,Y 333.646,Z 710.917,A -85,B 0,C 180,E1 -14702.596,E2 -14702.596} C_VEL
LIN {X 0,Y 333.679,Z 710.901,A -85,B 0,C 180,E1 -14706.14,E2 -14706.14} C_VEL
LIN {X 0,Y 333.635,Z 710.918,A -85,B 0,C 180,E1 -14707.845,E2 -14707.845} C_VEL
LIN {X 0,Y 332.934,Z 711.011,A -85,B 0,C 180,E1 -14708.853,E2 -14708.853} C_VEL
LIN {X 0,Y 330.079,Z 711.366,A -85,B 0,C 180,E1 -14710.492,E2 -14710.492} C_VEL
LIN {X 0,Y 327.678,Z 711.669,A -85,B 0,C 180,E1 -14711.82,E2 -14711.82} C_VEL
LIN {X 0,Y 326.645,Z 711.796,A -85,B 0,C 180,E1 -14712.848,E2 -14712.848} C_VEL
LIN {X 0,Y 326.558,Z 711.807,A -85,B 0,C 180,E1 -14713.196,E2 -14713.196} C_VEL
LIN {X 0,Y 326.577,Z 711.804,A -85,B 0,C 180,E1 -14717.03,E2 -14717.03} C_VEL
LIN {X 0,Y 326.578,Z 711.805,A -85,B 0,C 180,E1 -14720.782,E2 -14720.782} C_VEL
LIN {X 0,Y 326.698,Z 711.896,A -85,B 0,C 180,E1 -14724.663,E2 -14724.663} C_VEL
LIN {X 0,Y 326.829,Z 712.635,A -85,B 0,C 180,E1 -14724.869,E2 -14724.869} C_VEL
LIN {X 0,Y 334.242,Z 733.654,A -85,B 0,C 180,E1 -14725.876,E2 -14725.876} C_VEL
LIN {X 0,Y 332.955,Z 788.943,A -85,B 0,C 180,E1 -14727.364,E2 -14727.364} C_VEL
LIN {X 0,Y 332.7,Z 800.827,A -85,B 0,C 180,E1 -14727.865,E2 -14727.865} C_VEL
LIN {X 0,Y 332.285,Z 812.087,A -85,B 0,C 180,E1 -14728.523,E2 -14728.523} C_VEL
LIN {X 0,Y 331.796,Z 822.058,A -85,B 0,C 180,E1 -14729.269,E2 -14729.269} C_VEL
LIN {X 0,Y 331.21,Z 832.097,A -85,B 0,C 180,E1 -14730.199,E2 -14730.199} C_VEL
LIN {X 0,Y 330.655,Z 840.105,A -85,B 0,C 180,E1 -14731.082,E2 -14731.082} C_VEL
LIN {X 0,Y 329.984,Z 848.871,A -85,B 0,C 180,E1 -14732.232,E2 -14732.232} C_VEL
LIN {X 0,Y 329.437,Z 856.35,A -85,B 0,C 180,E1 -14733.384,E2 -14733.384} C_VEL
LIN {X 0,Y 328.855,Z 863.604,A -85,B 0,C 180,E1 -14734.696,E2 -14734.696} C_VEL
LIN {X 0,Y 328.131,Z 871.22,A -85,B 0,C 180,E1 -14736.355,E2 -14736.355} C_VEL
LIN {X 0,Y 327.695,Z 877.283,A -85,B 0,C 180,E1 -14737.956,E2 -14737.956} C_VEL
LIN {X 0,Y 327.379,Z 881.503,A -85,B 0,C 180,E1 -14739.254,E2 -14739.254} C_VEL
LIN {X 0,Y 327.011,Z 886.484,A -85,B 0,C 180,E1 -14741.193,E2 -14741.193} C_VEL
LIN {X 0,Y 326.817,Z 890.229,A -85,B 0,C 180,E1 -14743.123,E2 -14743.123} C_VEL
LIN {X 0,Y 326.713,Z 893.28,A -85,B 0,C 180,E1 -14745.473,E2 -14745.473} C_VEL
LIN {X 0,Y 326.779,Z 894.099,A -85,B 0,C 180,E1 -14746.315,E2 -14746.315} C_VEL
LIN {X 0,Y 326.864,Z 894.799,A -85,B 0,C 180,E1 -14747.583,E2 -14747.583} C_VEL
LIN {X 0,Y 327.061,Z 895.065,A -85,B 0,C 180,E1 -14748.849,E2 -14748.849} C_VEL
LIN {X 0,Y 327.306,Z 894.912,A -85,B 0,C 180,E1 -14750.109,E2 -14750.109} C_VEL
LIN {X 0,Y 327.929,Z 893.154,A -85,B 0,C 180,E1 -14752.612,E2 -14752.612} C_VEL
LIN {X 0,Y 328.393,Z 891.731,A -85,B 0,C 180,E1 -14753.857,E2 -14753.857} C_VEL
LIN {X 0,Y 329.176,Z 888.583,A -85,B 0,C 180,E1 -14755.714,E2 -14755.714} C_VEL
LIN {X 0,Y 330.261,Z 883.252,A -85,B 0,C 180,E1 -14757.935,E2 -14757.935} C_VEL
LIN {X 0,Y 331.139,Z 878.813,A -85,B 0,C 180,E1 -14759.392,E2 -14759.392} C_VEL
LIN {X 0,Y 332.259,Z 873.136,A -85,B 0,C 180,E1 -14760.909,E2 -14760.909} C_VEL
LIN {X 0,Y 333.404,Z 866.304,A -85,B 0,C 180,E1 -14762.416,E2 -14762.416} C_VEL
LIN {X 0,Y 334.46,Z 859.827,A -85,B 0,C 180,E1 -14763.614,E2 -14763.614} C_VEL
LIN {X 0,Y 335.684,Z 851.081,A -85,B 0,C 180,E1 -14764.954,E2 -14764.954} C_VEL
LIN {X 0,Y 336.694,Z 843.065,A -85,B 0,C 180,E1 -14765.991,E2 -14765.991} C_VEL
LIN {X 0,Y 337.693,Z 833.409,A -85,B 0,C 180,E1 -14767.023,E2 -14767.023} C_VEL
LIN {X 0,Y 338.527,Z 823.201,A -85,B 0,C 180,E1 -14767.905,E2 -14767.905} C_VEL
LIN {X 0,Y 339.171,Z 813.581,A -85,B 0,C 180,E1 -14768.565,E2 -14768.565} C_VEL
LIN {X 0,Y 339.628,Z 803.195,A -85,B 0,C 180,E1 -14769.116,E2 -14769.116} C_VEL
LIN {X 0,Y 339.877,Z 789.537,A -85,B 0,C 180,E1 -14769.637,E2 -14769.637} C_VEL
LIN {X 0,Y 341.287,Z 755.995,A -85,B 0,C 180,E1 -14770.648,E2 -14770.648} C_VEL
LIN {X 0,Y 342.142,Z 740.257,A -85,B 0,C 180,E1 -14771.115,E2 -14771.115} C_VEL
LIN {X 0,Y 336.384,Z 728.847,A -85,B 0,C 180,E1 -14772.271,E2 -14772.271} C_VEL
LIN {X 0,Y 330.83,Z 719.343,A -85,B 0,C 180,E1 -14773.438,E2 -14773.438} C_VEL
LIN {X 0,Y 328.917,Z 716.028,A -85,B 0,C 180,E1 -14773.869,E2 -14773.869} C_VEL
LIN {X 0,Y 327.209,Z 713.505,A -85,B 0,C 180,E1 -14774.25,E2 -14774.25} C_VEL
LIN {X 0,Y 326.817,Z 712.093,A -85,B 0,C 180,E1 -14774.51,E2 -14774.51} C_VEL
LIN {X 0,Y 326.761,Z 711.784,A -85,B 0,C 180,E1 -14774.957,E2 -14774.957} C_VEL
LIN {X 0,Y 326.715,Z 711.788,A -85,B 0,C 180,E1 -14778.824,E2 -14778.824} C_VEL
LIN {X 0,Y 326.61,Z 711.803,A -85,B 0,C 180,E1 -14782.788,E2 -14782.788} C_VEL
LIN {X 0,Y 326.651,Z 711.796,A -85,B 0,C 180,E1 -14785.487,E2 -14785.487} C_VEL
LIN {X 0,Y 326.635,Z 711.798,A -85,B 0,C 180,E1 -14788.253,E2 -14788.253} C_VEL
LIN {X 0,Y 326.582,Z 711.805,A -85,B 0,C 180,E1 -14791.096,E2 -14791.096} C_VEL
LIN {X 0,Y 326.614,Z 711.8,A -85,B 0,C 180,E1 -14794.019,E2 -14794.019} C_VEL
LIN {X 0,Y 326.634,Z 711.797,A -85,B 0,C 180,E1 -14797.238,E2 -14797.238} C_VEL
LIN {X 0,Y 326.584,Z 711.802,A -85,B 0,C 180,E1 -14801.13,E2 -14801.13} C_VEL
LIN {X 0,Y 326.534,Z 711.81,A -85,B 0,C 180,E1 -14804.742,E2 -14804.742} C_VEL
LIN {X 0,Y 326.582,Z 711.805,A -85,B 0,C 180,E1 -14808.153,E2 -14808.153} C_VEL
LIN {X 0,Y 326.642,Z 711.797,A -85,B 0,C 180,E1 -14812.131,E2 -14812.131} C_VEL
LIN {X 0,Y 326.667,Z 712.088,A -85,B 0,C 180,E1 -14812.501,E2 -14812.501} C_VEL
LIN {X 0,Y 330.084,Z 725.946,A -85,B 0,C 180,E1 -14815.821,E2 -14815.821} C_VEL
LIN {X 0,Y 333.107,Z 739.532,A -85,B 0,C 180,E1 -14818.873,E2 -14818.873} C_VEL
LIN {X 0,Y 333.583,Z 743.64,A -85,B 0,C 180,E1 -14819.746,E2 -14819.746} C_VEL
LIN {X 0,Y 331.638,Z 760.183,A -85,B 0,C 180,E1 -14822.905,E2 -14822.905} C_VEL
LIN {X 0,Y 334.343,Z 778.984,A -85,B 0,C 180,E1 -14824.009,E2 -14824.009} C_VEL
LIN {X 0,Y 337.013,Z 802.288,A -85,B 0,C 180,E1 -14825.187,E2 -14825.187} C_VEL
LIN {X 0,Y 338.649,Z 831.63,A -85,B 0,C 180,E1 -14826.392,E2 -14826.392} C_VEL
LIN {X 0,Y 336.487,Z 879.656,A -85,B 0,C 180,E1 -14827.809,E2 -14827.809} C_VEL
LIN {X 0,Y 335.71,Z 889.81,A -85,B 0,C 180,E1 -14828.225,E2 -14828.225} C_VEL
LIN {X 0,Y 334.84,Z 899.755,A -85,B 0,C 180,E1 -14828.771,E2 -14828.771} C_VEL
LIN {X 0,Y 333.585,Z 910.261,A -85,B 0,C 180,E1 -14829.495,E2 -14829.495} C_VEL
LIN {X 0,Y 332.241,Z 920.457,A -85,B 0,C 180,E1 -14830.376,E2 -14830.376} C_VEL
LIN {X 0,Y 330.871,Z 930.335,A -85,B 0,C 180,E1 -14831.419,E2 -14831.419} C_VEL
LIN {X 0,Y 329.744,Z 938.761,A -85,B 0,C 180,E1 -14832.477,E2 -14832.477} C_VEL
LIN {X 0,Y 328.306,Z 950.179,A -85,B 0,C 180,E1 -14834.159,E2 -14834.159} C_VEL
LIN {X 0,Y 327.352,Z 957.244,A -85,B 0,C 180,E1 -14835.387,E2 -14835.387} C_VEL
LIN {X 0,Y 326.613,Z 964.757,A -85,B 0,C 180,E1 -14836.94,E2 -14836.94} C_VEL
LIN {X 0,Y 325.971,Z 972.169,A -85,B 0,C 180,E1 -14838.809,E2 -14838.809} C_VEL
LIN {X 0,Y 325.716,Z 978.123,A -85,B 0,C 180,E1 -14840.685,E2 -14840.685} C_VEL
LIN {X 0,Y 325.679,Z 982.81,A -85,B 0,C 180,E1 -14842.559,E2 -14842.559} C_VEL
LIN {X 0,Y 325.788,Z 986.368,A -85,B 0,C 180,E1 -14844.427,E2 -14844.427} C_VEL
LIN {X 0,Y 326.017,Z 988.882,A -85,B 0,C 180,E1 -14846.29,E2 -14846.29} C_VEL
LIN {X 0,Y 326.081,Z 989.979,A -85,B 0,C 180,E1 -14847.528,E2 -14847.528} C_VEL
LIN {X 0,Y 326.174,Z 990.651,A -85,B 0,C 180,E1 -14848.764,E2 -14848.764} C_VEL
LIN {X 0,Y 326.257,Z 990.913,A -85,B 0,C 180,E1 -14849.998,E2 -14849.998} C_VEL
LIN {X 0,Y 326.16,Z 990.739,A -85,B 0,C 180,E1 -14851.233,E2 -14851.233} C_VEL
LIN {X 0,Y 326.062,Z 990.115,A -85,B 0,C 180,E1 -14852.469,E2 -14852.469} C_VEL
LIN {X 0,Y 326.013,Z 989.075,A -85,B 0,C 180,E1 -14853.706,E2 -14853.706} C_VEL
LIN {X 0,Y 325.866,Z 987.605,A -85,B 0,C 180,E1 -14854.947,E2 -14854.947} C_VEL
LIN {X 0,Y 325.692,Z 984.276,A -85,B 0,C 180,E1 -14856.964,E2 -14856.964} C_VEL
LIN {X 0,Y 325.616,Z 980.45,A -85,B 0,C 180,E1 -14858.688,E2 -14858.688} C_VEL
LIN {X 0,Y 325.859,Z 974.242,A -85,B 0,C 180,E1 -14860.876,E2 -14860.876} C_VEL
LIN {X 0,Y 326.452,Z 967.474,A -85,B 0,C 180,E1 -14862.746,E2 -14862.746} C_VEL
LIN {X 0,Y 327.403,Z 959.124,A -85,B 0,C 180,E1 -14864.607,E2 -14864.607} C_VEL
LIN {X 0,Y 328.495,Z 950.677,A -85,B 0,C 180,E1 -14866.147,E2 -14866.147} C_VEL
LIN {X 0,Y 329.642,Z 941.54,A -85,B 0,C 180,E1 -14867.524,E2 -14867.524} C_VEL
LIN {X 0,Y 331.29,Z 930.419,A -85,B 0,C 180,E1 -14868.873,E2 -14868.873} C_VEL
LIN {X 0,Y 332.867,Z 917.791,A -85,B 0,C 180,E1 -14870.063,E2 -14870.063} C_VEL
LIN {X 0,Y 334.252,Z 905.461,A -85,B 0,C 180,E1 -14870.941,E2 -14870.941} C_VEL
LIN {X 0,Y 335.413,Z 892.571,A -85,B 0,C 180,E1 -14871.59,E2 -14871.59} C_VEL
LIN {X 0,Y 336.003,Z 879.119,A -85,B 0,C 180,E1 -14872.034,E2 -14872.034} C_VEL
LIN {X 0,Y 337.035,Z 829.831,A -85,B 0,C 180,E1 -14873.122,E2 -14873.122} C_VEL
LIN {X 0,Y 333.981,Z 797.526,A -85,B 0,C 180,E1 -14874.129,E2 -14874.129} C_VEL
LIN {X 0,Y 330.669,Z 772.289,A -85,B 0,C 180,E1 -14875.035,E2 -14875.035} C_VEL
LIN {X 0,Y 330.88,Z 769.623,A -85,B 0,C 180,E1 -14875.473,E2 -14875.473} C_VEL
LIN {X 0,Y 333.719,Z 746.642,A -85,B 0,C 180,E1 -14880.009,E2 -14880.009} C_VEL
LIN {X 0,Y 333.948,Z 743.345,A -85,B 0,C 180,E1 -14880.684,E2 -14880.684} C_VEL
LIN {X 0,Y 331.872,Z 732.943,A -85,B 0,C 180,E1 -14883.088,E2 -14883.088} C_VEL
LIN {X 0,Y 329.301,Z 721.886,A -85,B 0,C 180,E1 -14885.806,E2 -14885.806} C_VEL
LIN {X 0,Y 326.633,Z 711.903,A -85,B 0,C 180,E1 -14888.493,E2 -14888.493} C_VEL
LIN {X 0,Y 326.569,Z 711.808,A -85,B 0,C 180,E1 -14891.844,E2 -14891.844} C_VEL
LIN {X 0,Y 326.548,Z 711.805,A -85,B 0,C 180,E1 -14895.251,E2 -14895.251} C_VEL
LIN {X 0,Y 326.569,Z 711.801,A -85,B 0,C 180,E1 -14898.867,E2 -14898.867} C_VEL
LIN {X 0,Y 326.62,Z 711.799,A -85,B 0,C 180,E1 -14902.76,E2 -14902.76} C_VEL
LIN {X 0,Y 326.598,Z 711.796,A -85,B 0,C 180,E1 -14905.98,E2 -14905.98} C_VEL
LIN {X 0,Y 326.65,Z 711.796,A -85,B 0,C 180,E1 -14910.34,E2 -14910.34} C_VEL
LIN {X 0,Y 326.679,Z 711.789,A -85,B 0,C 180,E1 -14914.515,E2 -14914.515} C_VEL
LIN {X 0,Y 326.635,Z 711.79,A -85,B 0,C 180,E1 -14918.545,E2 -14918.545} C_VEL
LIN {X 0,Y 326.733,Z 711.786,A -85,B 0,C 180,E1 -14921.177,E2 -14921.177} C_VEL
LIN {X 0,Y 326.751,Z 711.784,A -85,B 0,C 180,E1 -14925.432,E2 -14925.432} C_VEL
LIN {X 0,Y 326.758,Z 711.781,A -85,B 0,C 180,E1 -14928.839,E2 -14928.839} C_VEL
LIN {X 0,Y 326.946,Z 711.759,A -85,B 0,C 180,E1 -14932.59,E2 -14932.59} C_VEL
LIN {X 0,Y 326.766,Z 711.774,A -85,B 0,C 180,E1 -14935.065,E2 -14935.065} C_VEL
LIN {X 0,Y 327.037,Z 711.745,A -85,B 0,C 180,E1 -14937.537,E2 -14937.537} C_VEL
LIN {X 0,Y 327.186,Z 711.721,A -85,B 0,C 180,E1 -14940,E2 -14940} C_VEL
LIN {X 0,Y 327.036,Z 711.75,A -85,B 0,C 180,E1 -14942.464,E2 -14942.464} C_VEL
LIN {X 0,Y 326.957,Z 711.753,A -85,B 0,C 180,E1 -14946.724,E2 -14946.724} C_VEL
LIN {X 0,Y 326.802,Z 711.774,A -85,B 0,C 180,E1 -14949.907,E2 -14949.907} C_VEL
LIN {X 0,Y 326.748,Z 711.783,A -85,B 0,C 180,E1 -14953.686,E2 -14953.686} C_VEL
LIN {X 0,Y 326.688,Z 711.792,A -85,B 0,C 180,E1 -14957.529,E2 -14957.529} C_VEL
LIN {X 0,Y 326.647,Z 711.794,A -85,B 0,C 180,E1 -14960.136,E2 -14960.136} C_VEL
LIN {X 0,Y 326.638,Z 711.78,A -85,B 0,C 180,E1 -14964.13,E2 -14964.13} C_VEL
LIN {X 0,Y 326.672,Z 711.794,A -85,B 0,C 180,E1 -14966.859,E2 -14966.859} C_VEL
LIN {X 0,Y 326.625,Z 711.802,A -85,B 0,C 180,E1 -14970.611,E2 -14970.611} C_VEL
LIN {X 0,Y 326.599,Z 711.802,A -85,B 0,C 180,E1 -14974.021,E2 -14974.021} C_VEL
LIN {X 0,Y 326.621,Z 711.801,A -85,B 0,C 180,E1 -14977.241,E2 -14977.241} C_VEL
LIN {X 0,Y 326.641,Z 712.002,A -85,B 0,C 180,E1 -14979.998,E2 -14979.998} C_VEL
LIN {X 0,Y 326.872,Z 713.059,A -85,B 0,C 180,E1 -14980.213,E2 -14980.213} C_VEL
LIN {X 0,Y 335.075,Z 729.716,A -85,B 0,C 180,E1 -14981.385,E2 -14981.385} C_VEL
LIN {X 0,Y 338.77,Z 738.225,A -85,B 0,C 180,E1 -14981.903,E2 -14981.903} C_VEL
LIN {X 0,Y 337.949,Z 792.147,A -85,B 0,C 180,E1 -14983.136,E2 -14983.136} C_VEL
LIN {X 0,Y 337.752,Z 805.344,A -85,B 0,C 180,E1 -14983.606,E2 -14983.606} C_VEL
LIN {X 0,Y 337.398,Z 817.473,A -85,B 0,C 180,E1 -14984.275,E2 -14984.275} C_VEL
LIN {X 0,Y 336.709,Z 828.786,A -85,B 0,C 180,E1 -14985.119,E2 -14985.119} C_VEL
LIN {X 0,Y 335.769,Z 839.374,A -85,B 0,C 180,E1 -14986.128,E2 -14986.128} C_VEL
LIN {X 0,Y 334.618,Z 850.35,A -85,B 0,C 180,E1 -14987.453,E2 -14987.453} C_VEL
LIN {X 0,Y 333.314,Z 860.484,A -85,B 0,C 180,E1 -14988.986,E2 -14988.986} C_VEL
LIN {X 0,Y 332.08,Z 868.973,A -85,B 0,C 180,E1 -14990.59,E2 -14990.59} C_VEL
LIN {X 0,Y 330.881,Z 876.575,A -85,B 0,C 180,E1 -14992.366,E2 -14992.366} C_VEL
LIN {X 0,Y 329.958,Z 882.329,A -85,B 0,C 180,E1 -14994.037,E2 -14994.037} C_VEL
LIN {X 0,Y 328.835,Z 888.296,A -85,B 0,C 180,E1 -14996.245,E2 -14996.245} C_VEL
LIN {X 0,Y 328.117,Z 892.415,A -85,B 0,C 180,E1 -14998.35,E2 -14998.35} C_VEL
LIN {X 0,Y 327.551,Z 895.224,A -85,B 0,C 180,E1 -15000.432,E2 -15000.432} C_VEL
LIN {X 0,Y 327.311,Z 896.452,A -85,B 0,C 180,E1 -15001.813,E2 -15001.813} C_VEL
LIN {X 0,Y 327.108,Z 897.135,A -85,B 0,C 180,E1 -15003.182,E2 -15003.182} C_VEL
LIN {X 0,Y 327.012,Z 897.365,A -85,B 0,C 180,E1 -15004.545,E2 -15004.545} C_VEL
LIN {X 0,Y 326.919,Z 897.129,A -85,B 0,C 180,E1 -15005.894,E2 -15005.894} C_VEL
LIN {X 0,Y 327.006,Z 896.185,A -85,B 0,C 180,E1 -15007.542,E2 -15007.542} C_VEL
LIN {X 0,Y 327.397,Z 893.56,A -85,B 0,C 180,E1 -15009.914,E2 -15009.914} C_VEL
LIN {X 0,Y 327.853,Z 890.18,A -85,B 0,C 180,E1 -15011.893,E2 -15011.893} C_VEL
LIN {X 0,Y 328.479,Z 885.642,A -85,B 0,C 180,E1 -15013.853,E2 -15013.853} C_VEL
LIN {X 0,Y 329.279,Z 879.831,A -85,B 0,C 180,E1 -15015.793,E2 -15015.793} C_VEL
LIN {X 0,Y 330.266,Z 872.541,A -85,B 0,C 180,E1 -15017.716,E2 -15017.716} C_VEL
LIN {X 0,Y 331.217,Z 865.07,A -85,B 0,C 180,E1 -15019.302,E2 -15019.302} C_VEL
LIN {X 0,Y 332.281,Z 856.011,A -85,B 0,C 180,E1 -15020.874,E2 -15020.874} C_VEL
LIN {X 0,Y 333.329,Z 845.939,A -85,B 0,C 180,E1 -15022.295,E2 -15022.295} C_VEL
LIN {X 0,Y 334.29,Z 835.171,A -85,B 0,C 180,E1 -15023.513,E2 -15023.513} C_VEL
LIN {X 0,Y 335.201,Z 822.912,A -85,B 0,C 180,E1 -15024.588,E2 -15024.588} C_VEL
LIN {X 0,Y 335.704,Z 810.413,A -85,B 0,C 180,E1 -15025.424,E2 -15025.424} C_VEL
LIN {X 0,Y 336.013,Z 797.237,A -85,B 0,C 180,E1 -15026.029,E2 -15026.029} C_VEL
LIN {X 0,Y 336.152,Z 779.392,A -85,B 0,C 180,E1 -15026.501,E2 -15026.501} C_VEL
LIN {X 0,Y 336.799,Z 735.869,A -85,B 0,C 180,E1 -15027.464,E2 -15027.464} C_VEL
LIN {X 0,Y 327.662,Z 713.933,A -85,B 0,C 180,E1 -15028.631,E2 -15028.631} C_VEL
LIN {X 0,Y 327.088,Z 712.207,A -85,B 0,C 180,E1 -15028.809,E2 -15028.809} C_VEL
LIN {X 0,Y 327.022,Z 711.786,A -85,B 0,C 180,E1 -15029.078,E2 -15029.078} C_VEL
LIN {X 0,Y 327.004,Z 711.751,A -85,B 0,C 180,E1 -15032.465,E2 -15032.465} C_VEL
LIN {X 0,Y 326.944,Z 711.761,A -85,B 0,C 180,E1 -15036.172,E2 -15036.172} C_VEL
LIN {X 0,Y 326.785,Z 711.776,A -85,B 0,C 180,E1 -15039.909,E2 -15039.909} C_VEL
LIN {X 0,Y 326.761,Z 711.779,A -85,B 0,C 180,E1 -15043.687,E2 -15043.687} C_VEL
LIN {X 0,Y 326.659,Z 711.794,A -85,B 0,C 180,E1 -15047.532,E2 -15047.532} C_VEL
LIN {X 0,Y 326.614,Z 711.796,A -85,B 0,C 180,E1 -15051.459,E2 -15051.459} C_VEL
LIN {X 0,Y 326.606,Z 711.785,A -85,B 0,C 180,E1 -15055.493,E2 -15055.493} C_VEL
LIN {X 0,Y 326.595,Z 711.792,A -85,B 0,C 180,E1 -15058.258,E2 -15058.258} C_VEL
LIN {X 0,Y 326.574,Z 711.806,A -85,B 0,C 180,E1 -15061.099,E2 -15061.099} C_VEL
LIN {X 0,Y 326.612,Z 711.775,A -85,B 0,C 180,E1 -15064.021,E2 -15064.021} C_VEL
LIN {X 0,Y 326.581,Z 711.792,A -85,B 0,C 180,E1 -15067.835,E2 -15067.835} C_VEL
LIN {X 0,Y 326.554,Z 711.809,A -85,B 0,C 180,E1 -15071.851,E2 -15071.851} C_VEL
LIN {X 0,Y 326.558,Z 711.807,A -85,B 0,C 180,E1 -15073.196,E2 -15073.196} C_VEL
LIN {X 0,Y 325.883,Z 711.896,A -85,B 0,C 180,E1 -15074.226,E2 -15074.226} C_VEL
LIN {X 0,Y 323.031,Z 712.251,A -85,B 0,C 180,E1 -15075.903,E2 -15075.903} C_VEL
LIN {X 0,Y 320.621,Z 712.547,A -85,B 0,C 180,E1 -15077.261,E2 -15077.261} C_VEL
LIN {X 0,Y 319.588,Z 712.675,A -85,B 0,C 180,E1 -15078.313,E2 -15078.313} C_VEL
LIN {X 0,Y 319.505,Z 712.685,A -85,B 0,C 180,E1 -15078.669,E2 -15078.669} C_VEL
LIN {X 0,Y 319.547,Z 712.681,A -85,B 0,C 180,E1 -15082.354,E2 -15082.354} C_VEL
LIN {X 0,Y 319.642,Z 712.906,A -85,B 0,C 180,E1 -15084.371,E2 -15084.371} C_VEL
LIN {X 0,Y 319.891,Z 713.85,A -85,B 0,C 180,E1 -15084.554,E2 -15084.554} C_VEL
LIN {X 0,Y 327.399,Z 735.146,A -85,B 0,C 180,E1 -15085.585,E2 -15085.585} C_VEL
LIN {X 0,Y 326.088,Z 787.905,A -85,B 0,C 180,E1 -15087.022,E2 -15087.022} C_VEL
LIN {X 0,Y 325.815,Z 801.52,A -85,B 0,C 180,E1 -15087.595,E2 -15087.595} C_VEL
LIN {X 0,Y 325.39,Z 812.366,A -85,B 0,C 180,E1 -15088.232,E2 -15088.232} C_VEL
LIN {X 0,Y 324.957,Z 821.529,A -85,B 0,C 180,E1 -15088.911,E2 -15088.911} C_VEL
LIN {X 0,Y 324.298,Z 832.438,A -85,B 0,C 180,E1 -15089.923,E2 -15089.923} C_VEL
LIN {X 0,Y 323.664,Z 841.395,A -85,B 0,C 180,E1 -15090.932,E2 -15090.932} C_VEL
LIN {X 0,Y 322.965,Z 850.127,A -85,B 0,C 180,E1 -15092.104,E2 -15092.104} C_VEL
LIN {X 0,Y 322.392,Z 857.973,A -85,B 0,C 180,E1 -15093.356,E2 -15093.356} C_VEL
LIN {X 0,Y 321.748,Z 865.576,A -85,B 0,C 180,E1 -15094.789,E2 -15094.789} C_VEL
LIN {X 0,Y 321.163,Z 871.619,A -85,B 0,C 180,E1 -15096.119,E2 -15096.119} C_VEL
LIN {X 0,Y 320.745,Z 877.026,A -85,B 0,C 180,E1 -15097.516,E2 -15097.516} C_VEL
LIN {X 0,Y 320.282,Z 883.083,A -85,B 0,C 180,E1 -15099.446,E2 -15099.446} C_VEL
LIN {X 0,Y 319.948,Z 887.953,A -85,B 0,C 180,E1 -15101.427,E2 -15101.427} C_VEL
LIN {X 0,Y 319.822,Z 890.605,A -85,B 0,C 180,E1 -15102.743,E2 -15102.743} C_VEL
LIN {X 0,Y 319.707,Z 893.505,A -85,B 0,C 180,E1 -15104.705,E2 -15104.705} C_VEL
LIN {X 0,Y 319.839,Z 895.729,A -85,B 0,C 180,E1 -15107.306,E2 -15107.306} C_VEL
LIN {X 0,Y 320.016,Z 896.154,A -85,B 0,C 180,E1 -15108.6,E2 -15108.6} C_VEL
LIN {X 0,Y 320.461,Z 895.842,A -85,B 0,C 180,E1 -15110.721,E2 -15110.721} C_VEL
LIN {X 0,Y 320.911,Z 894.768,A -85,B 0,C 180,E1 -15112.449,E2 -15112.449} C_VEL
LIN {X 0,Y 321.367,Z 893.407,A -85,B 0,C 180,E1 -15113.722,E2 -15113.722} C_VEL
LIN {X 0,Y 322.468,Z 889.349,A -85,B 0,C 180,E1 -15116.251,E2 -15116.251} C_VEL
LIN {X 0,Y 323.468,Z 884.976,A -85,B 0,C 180,E1 -15118.133,E2 -15118.133} C_VEL
LIN {X 0,Y 324.453,Z 880.408,A -85,B 0,C 180,E1 -15119.69,E2 -15119.69} C_VEL
LIN {X 0,Y 325.628,Z 874.808,A -85,B 0,C 180,E1 -15121.237,E2 -15121.237} C_VEL
LIN {X 0,Y 326.852,Z 868.08,A -85,B 0,C 180,E1 -15122.773,E2 -15122.773} C_VEL
LIN {X 0,Y 328.246,Z 859.92,A -85,B 0,C 180,E1 -15124.297,E2 -15124.297} C_VEL
LIN {X 0,Y 329.436,Z 852.118,A -85,B 0,C 180,E1 -15125.509,E2 -15125.509} C_VEL
LIN {X 0,Y 330.49,Z 844.066,A -85,B 0,C 180,E1 -15126.563,E2 -15126.563} C_VEL
LIN {X 0,Y 331.548,Z 834.345,A -85,B 0,C 180,E1 -15127.613,E2 -15127.613} C_VEL
LIN {X 0,Y 332.333,Z 825.975,A -85,B 0,C 180,E1 -15128.36,E2 -15128.36} C_VEL
LIN {X 0,Y 333.02,Z 815.698,A -85,B 0,C 180,E1 -15129.107,E2 -15129.107} C_VEL
LIN {X 0,Y 333.605,Z 804.877,A -85,B 0,C 180,E1 -15129.702,E2 -15129.702} C_VEL
LIN {X 0,Y 333.891,Z 791.878,A -85,B 0,C 180,E1 -15130.23,E2 -15130.23} C_VEL
LIN {X 0,Y 334.973,Z 766.363,A -85,B 0,C 180,E1 -15131.026,E2 -15131.026} C_VEL
LIN {X 0,Y 336.306,Z 742.672,A -85,B 0,C 180,E1 -15131.747,E2 -15131.747} C_VEL
LIN {X 0,Y 330.749,Z 731.607,A -85,B 0,C 180,E1 -15132.944,E2 -15132.944} C_VEL
LIN {X 0,Y 324.561,Z 721.079,A -85,B 0,C 180,E1 -15134.337,E2 -15134.337} C_VEL
LIN {X 0,Y 321.9,Z 716.957,A -85,B 0,C 180,E1 -15134.965,E2 -15134.965} C_VEL
LIN {X 0,Y 320.192,Z 714.49,A -85,B 0,C 180,E1 -15135.378,E2 -15135.378} C_VEL
LIN {X 0,Y 319.739,Z 713.019,A -85,B 0,C 180,E1 -15135.661,E2 -15135.661} C_VEL
LIN {X 0,Y 319.698,Z 712.712,A -85,B 0,C 180,E1 -15135.884,E2 -15135.884} C_VEL
LIN {X 0,Y 319.641,Z 712.67,A -85,B 0,C 180,E1 -15139.257,E2 -15139.257} C_VEL
LIN {X 0,Y 319.565,Z 712.677,A -85,B 0,C 180,E1 -15143.32,E2 -15143.32} C_VEL
LIN {X 0,Y 319.586,Z 712.678,A -85,B 0,C 180,E1 -15146.092,E2 -15146.092} C_VEL
LIN {X 0,Y 319.565,Z 712.678,A -85,B 0,C 180,E1 -15148.936,E2 -15148.936} C_VEL
LIN {X 0,Y 319.532,Z 712.683,A -85,B 0,C 180,E1 -15151.862,E2 -15151.862} C_VEL
LIN {X 0,Y 319.587,Z 712.678,A -85,B 0,C 180,E1 -15155.542,E2 -15155.542} C_VEL
LIN {X 0,Y 319.58,Z 712.677,A -85,B 0,C 180,E1 -15158.007,E2 -15158.007} C_VEL
LIN {X 0,Y 319.532,Z 712.682,A -85,B 0,C 180,E1 -15161.596,E2 -15161.596} C_VEL
LIN {X 0,Y 319.495,Z 712.686,A -85,B 0,C 180,E1 -15165.256,E2 -15165.256} C_VEL
LIN {X 0,Y 319.534,Z 712.681,A -85,B 0,C 180,E1 -15168.711,E2 -15168.711} C_VEL
LIN {X 0,Y 319.631,Z 712.892,A -85,B 0,C 180,E1 -15172.02,E2 -15172.02} C_VEL
LIN {X 0,Y 322.889,Z 726.237,A -85,B 0,C 180,E1 -15175.3,E2 -15175.3} C_VEL
LIN {X 0,Y 325.956,Z 739.942,A -85,B 0,C 180,E1 -15178.474,E2 -15178.474} C_VEL
LIN {X 0,Y 326.645,Z 744.08,A -85,B 0,C 180,E1 -15179.387,E2 -15179.387} C_VEL
LIN {X 0,Y 325.178,Z 756.598,A -85,B 0,C 180,E1 -15181.841,E2 -15181.841} C_VEL
LIN {X 0,Y 327.771,Z 774.268,A -85,B 0,C 180,E1 -15182.974,E2 -15182.974} C_VEL
LIN {X 0,Y 330.272,Z 795.073,A -85,B 0,C 180,E1 -15184.119,E2 -15184.119} C_VEL
LIN {X 0,Y 331.408,Z 808.468,A -85,B 0,C 180,E1 -15184.762,E2 -15184.762} C_VEL
LIN {X 0,Y 332.568,Z 832.607,A -85,B 0,C 180,E1 -15185.783,E2 -15185.783} C_VEL
LIN {X 0,Y 330.305,Z 878.976,A -85,B 0,C 180,E1 -15187.196,E2 -15187.196} C_VEL
LIN {X 0,Y 329.351,Z 890.44,A -85,B 0,C 180,E1 -15187.7,E2 -15187.7} C_VEL
LIN {X 0,Y 327.915,Z 904.409,A -85,B 0,C 180,E1 -15188.548,E2 -15188.548} C_VEL
LIN {X 0,Y 326.069,Z 917.782,A -85,B 0,C 180,E1 -15189.66,E2 -15189.66} C_VEL
LIN {X 0,Y 324.534,Z 927.859,A -85,B 0,C 180,E1 -15190.714,E2 -15190.714} C_VEL
LIN {X 0,Y 323.204,Z 936.381,A -85,B 0,C 180,E1 -15191.783,E2 -15191.783} C_VEL
LIN {X 0,Y 321.779,Z 945.604,A -85,B 0,C 180,E1 -15193.176,E2 -15193.176} C_VEL
LIN {X 0,Y 320.615,Z 954.35,A -85,B 0,C 180,E1 -15194.747,E2 -15194.747} C_VEL
LIN {X 0,Y 319.793,Z 962.198,A -85,B 0,C 180,E1 -15196.333,E2 -15196.333} C_VEL
LIN {X 0,Y 319.067,Z 969.881,A -85,B 0,C 180,E1 -15198.242,E2 -15198.242} C_VEL
LIN {X 0,Y 318.651,Z 977.006,A -85,B 0,C 180,E1 -15200.477,E2 -15200.477} C_VEL
LIN {X 0,Y 318.618,Z 981.722,A -85,B 0,C 180,E1 -15202.393,E2 -15202.393} C_VEL
LIN {X 0,Y 318.712,Z 985.298,A -85,B 0,C 180,E1 -15204.303,E2 -15204.303} C_VEL
LIN {X 0,Y 318.973,Z 987.833,A -85,B 0,C 180,E1 -15206.208,E2 -15206.208} C_VEL
LIN {X 0,Y 319.039,Z 988.948,A -85,B 0,C 180,E1 -15207.473,E2 -15207.473} C_VEL
LIN {X 0,Y 319.138,Z 989.629,A -85,B 0,C 180,E1 -15208.736,E2 -15208.736} C_VEL
LIN {X 0,Y 319.228,Z 989.898,A -85,B 0,C 180,E1 -15209.998,E2 -15209.998} C_VEL
LIN {X 0,Y 319.123,Z 989.731,A -85,B 0,C 180,E1 -15211.26,E2 -15211.26} C_VEL
LIN {X 0,Y 319.016,Z 989.12,A -85,B 0,C 180,E1 -15212.523,E2 -15212.523} C_VEL
LIN {X 0,Y 318.967,Z 988.085,A -85,B 0,C 180,E1 -15213.788,E2 -15213.788} C_VEL
LIN {X 0,Y 318.795,Z 986.616,A -85,B 0,C 180,E1 -15215.057,E2 -15215.057} C_VEL
LIN {X 0,Y 318.627,Z 983.54,A -85,B 0,C 180,E1 -15216.987,E2 -15216.987} C_VEL
LIN {X 0,Y 318.537,Z 979.482,A -85,B 0,C 180,E1 -15218.883,E2 -15218.883} C_VEL
LIN {X 0,Y 318.832,Z 973.298,A -85,B 0,C 180,E1 -15221.119,E2 -15221.119} C_VEL
LIN {X 0,Y 319.457,Z 966.565,A -85,B 0,C 180,E1 -15223.03,E2 -15223.03} C_VEL
LIN {X 0,Y 320.378,Z 958.834,A -85,B 0,C 180,E1 -15224.812,E2 -15224.812} C_VEL
LIN {X 0,Y 321.58,Z 949.848,A -85,B 0,C 180,E1 -15226.504,E2 -15226.504} C_VEL
LIN {X 0,Y 322.88,Z 940.765,A -85,B 0,C 180,E1 -15227.904,E2 -15227.904} C_VEL
LIN {X 0,Y 324.542,Z 929.719,A -85,B 0,C 180,E1 -15229.281,E2 -15229.281} C_VEL
LIN {X 0,Y 326.193,Z 917.189,A -85,B 0,C 180,E1 -15230.492,E2 -15230.492} C_VEL
LIN {X 0,Y 327.631,Z 904.987,A -85,B 0,C 180,E1 -15231.385,E2 -15231.385} C_VEL
LIN {X 0,Y 328.806,Z 892.453,A -85,B 0,C 180,E1 -15232.046,E2 -15232.046} C_VEL
LIN {X 0,Y 329.463,Z 879.598,A -85,B 0,C 180,E1 -15232.495,E2 -15232.495} C_VEL
LIN {X 0,Y 330.499,Z 829.67,A -85,B 0,C 180,E1 -15233.631,E2 -15233.631} C_VEL
LIN {X 0,Y 327.564,Z 798.369,A -85,B 0,C 180,E1 -15234.639,E2 -15234.639} C_VEL
LIN {X 0,Y 324.071,Z 772.057,A -85,B 0,C 180,E1 -15235.604,E2 -15235.604} C_VEL
LIN {X 0,Y 323.98,Z 770.543,A -85,B 0,C 180,E1 -15235.71,E2 -15235.71} C_VEL
LIN {X 0,Y 326.893,Z 747.919,A -85,B 0,C 180,E1 -15240.258,E2 -15240.258} C_VEL
LIN {X 0,Y 326.992,Z 744.206,A -85,B 0,C 180,E1 -15241.051,E2 -15241.051} C_VEL
LIN {X 0,Y 324.606,Z 732.369,A -85,B 0,C 180,E1 -15243.881,E2 -15243.881} C_VEL
LIN {X 0,Y 321.55,Z 719.955,A -85,B 0,C 180,E1 -15247.083,E2 -15247.083} C_VEL
LIN {X 0,Y 319.587,Z 712.773,A -85,B 0,C 180,E1 -15249.127,E2 -15249.127} C_VEL
LIN {X 0,Y 319.55,Z 712.674,A -85,B 0,C 180,E1 -15253.466,E2 -15253.466} C_VEL
LIN {X 0,Y 319.552,Z 712.674,A -85,B 0,C 180,E1 -15257.016,E2 -15257.016} C_VEL
LIN {X 0,Y 319.538,Z 712.668,A -85,B 0,C 180,E1 -15260.37,E2 -15260.37} C_VEL
LIN {X 0,Y 319.55,Z 712.67,A -85,B 0,C 180,E1 -15263.571,E2 -15263.571} C_VEL
LIN {X 0,Y 319.567,Z 712.676,A -85,B 0,C 180,E1 -15266.685,E2 -15266.685} C_VEL
LIN {X 0,Y 319.581,Z 712.678,A -85,B 0,C 180,E1 -15269.616,E2 -15269.616} C_VEL
LIN {X 0,Y 319.598,Z 712.671,A -85,B 0,C 180,E1 -15272.497,E2 -15272.497} C_VEL
LIN {X 0,Y 319.594,Z 712.67,A -85,B 0,C 180,E1 -15275.303,E2 -15275.303} C_VEL
LIN {X 0,Y 319.586,Z 712.67,A -85,B 0,C 180,E1 -15278.047,E2 -15278.047} C_VEL
LIN {X 0,Y 319.678,Z 712.664,A -85,B 0,C 180,E1 -15280.961,E2 -15280.961} C_VEL
LIN {X 0,Y 319.719,Z 712.659,A -85,B 0,C 180,E1 -15285.275,E2 -15285.275} C_VEL
LIN {X 0,Y 319.74,Z 712.653,A -85,B 0,C 180,E1 -15289.872,E2 -15289.872} C_VEL
LIN {X 0,Y 319.9,Z 712.634,A -85,B 0,C 180,E1 -15292.426,E2 -15292.426} C_VEL
LIN {X 0,Y 319.735,Z 712.65,A -85,B 0,C 180,E1 -15294.956,E2 -15294.956} C_VEL
LIN {X 0,Y 319.98,Z 712.624,A -85,B 0,C 180,E1 -15297.483,E2 -15297.483} C_VEL
LIN {X 0,Y 320.138,Z 712.599,A -85,B 0,C 180,E1 -15300,E2 -15300} C_VEL
LIN {X 0,Y 319.979,Z 712.628,A -85,B 0,C 180,E1 -15302.518,E2 -15302.518} C_VEL
LIN {X 0,Y 319.916,Z 712.631,A -85,B 0,C 180,E1 -15306.716,E2 -15306.716} C_VEL
LIN {X 0,Y 319.746,Z 712.654,A -85,B 0,C 180,E1 -15310.128,E2 -15310.128} C_VEL
LIN {X 0,Y 319.72,Z 712.66,A -85,B 0,C 180,E1 -15314.725,E2 -15314.725} C_VEL
LIN {X 0,Y 319.678,Z 712.66,A -85,B 0,C 180,E1 -15319.039,E2 -15319.039} C_VEL
LIN {X 0,Y 319.549,Z 712.661,A -85,B 0,C 180,E1 -15323.321,E2 -15323.321} C_VEL
LIN {X 0,Y 319.624,Z 712.674,A -85,B 0,C 180,E1 -15326.089,E2 -15326.089} C_VEL
LIN {X 0,Y 319.57,Z 712.664,A -85,B 0,C 180,E1 -15328.936,E2 -15328.936} C_VEL
LIN {X 0,Y 319.523,Z 712.677,A -85,B 0,C 180,E1 -15331.863,E2 -15331.863} C_VEL
LIN {X 0,Y 319.572,Z 712.671,A -85,B 0,C 180,E1 -15335.545,E2 -15335.545} C_VEL
LIN {X 0,Y 319.605,Z 712.835,A -85,B 0,C 180,E1 -15339.315,E2 -15339.315} C_VEL
LIN {X 0,Y 319.833,Z 713.922,A -85,B 0,C 180,E1 -15339.557,E2 -15339.557} C_VEL
LIN {X 0,Y 329.333,Z 733.075,A -85,B 0,C 180,E1 -15340.963,E2 -15340.963} C_VEL
LIN {X 0,Y 332.472,Z 740.401,A -85,B 0,C 180,E1 -15341.424,E2 -15341.424} C_VEL
LIN {X 0,Y 331.492,Z 790.268,A -85,B 0,C 180,E1 -15342.567,E2 -15342.567} C_VEL
LIN {X 0,Y 331.397,Z 803.554,A -85,B 0,C 180,E1 -15343.001,E2 -15343.001} C_VEL
LIN {X 0,Y 331.057,Z 815.565,A -85,B 0,C 180,E1 -15343.625,E2 -15343.625} C_VEL
LIN {X 0,Y 330.399,Z 827.183,A -85,B 0,C 180,E1 -15344.449,E2 -15344.449} C_VEL
LIN {X 0,Y 329.439,Z 838.311,A -85,B 0,C 180,E1 -15345.469,E2 -15345.469} C_VEL
LIN {X 0,Y 328.263,Z 849.275,A -85,B 0,C 180,E1 -15346.759,E2 -15346.759} C_VEL
LIN {X 0,Y 326.976,Z 859.195,A -85,B 0,C 180,E1 -15348.22,E2 -15348.22} C_VEL
LIN {X 0,Y 325.799,Z 867.252,A -85,B 0,C 180,E1 -15349.676,E2 -15349.676} C_VEL
LIN {X 0,Y 324.442,Z 875.562,A -85,B 0,C 180,E1 -15351.52,E2 -15351.52} C_VEL
LIN {X 0,Y 323.221,Z 882.746,A -85,B 0,C 180,E1 -15353.564,E2 -15353.564} C_VEL
LIN {X 0,Y 322.2,Z 887.977,A -85,B 0,C 180,E1 -15355.452,E2 -15355.452} C_VEL
LIN {X 0,Y 321.35,Z 892.497,A -85,B 0,C 180,E1 -15357.603,E2 -15357.603} C_VEL
LIN {X 0,Y 320.703,Z 895.649,A -85,B 0,C 180,E1 -15359.735,E2 -15359.735} C_VEL
LIN {X 0,Y 320.383,Z 897.181,A -85,B 0,C 180,E1 -15361.337,E2 -15361.337} C_VEL
LIN {X 0,Y 320.17,Z 897.947,A -85,B 0,C 180,E1 -15362.553,E2 -15362.553} C_VEL
LIN {X 0,Y 320.015,Z 898.362,A -85,B 0,C 180,E1 -15364.214,E2 -15364.214} C_VEL
LIN {X 0,Y 319.929,Z 897.77,A -85,B 0,C 180,E1 -15366.711,E2 -15366.711} C_VEL
LIN {X 0,Y 320.04,Z 896.749,A -85,B 0,C 180,E1 -15368.082,E2 -15368.082} C_VEL
LIN {X 0,Y 320.491,Z 893.74,A -85,B 0,C 180,E1 -15370.553,E2 -15370.553} C_VEL
LIN {X 0,Y 321.135,Z 889.491,A -85,B 0,C 180,E1 -15372.818,E2 -15372.818} C_VEL
LIN {X 0,Y 321.86,Z 884.44,A -85,B 0,C 180,E1 -15374.812,E2 -15374.812} C_VEL
LIN {X 0,Y 322.748,Z 878.056,A -85,B 0,C 180,E1 -15376.785,E2 -15376.785} C_VEL
LIN {X 0,Y 323.841,Z 870.082,A -85,B 0,C 180,E1 -15378.739,E2 -15378.739} C_VEL
LIN {X 0,Y 324.863,Z 861.897,A -85,B 0,C 180,E1 -15380.35,E2 -15380.35} C_VEL
LIN {X 0,Y 325.992,Z 852.182,A -85,B 0,C 180,E1 -15381.906,E2 -15381.906} C_VEL
LIN {X 0,Y 327.033,Z 842.099,A -85,B 0,C 180,E1 -15383.214,E2 -15383.214} C_VEL
LIN {X 0,Y 327.976,Z 831.536,A -85,B 0,C 180,E1 -15384.314,E2 -15384.314} C_VEL
LIN {X 0,Y 328.696,Z 820.1,A -85,B 0,C 180,E1 -15385.249,E2 -15385.249} C_VEL
LIN {X 0,Y 329.196,Z 807.432,A -85,B 0,C 180,E1 -15386.023,E2 -15386.023} C_VEL
LIN {X 0,Y 329.444,Z 794.461,A -85,B 0,C 180,E1 -15386.562,E2 -15386.562} C_VEL
LIN {X 0,Y 330.092,Z 746.506,A -85,B 0,C 180,E1 -15387.676,E2 -15387.676} C_VEL
LIN {X 0,Y 330.285,Z 737.831,A -85,B 0,C 180,E1 -15387.868,E2 -15387.868} C_VEL
LIN {X 0,Y 321.648,Z 717.077,A -85,B 0,C 180,E1 -15388.997,E2 -15388.997} C_VEL
LIN {X 0,Y 320.147,Z 713.501,A -85,B 0,C 180,E1 -15389.239,E2 -15389.239} C_VEL
LIN {X 0,Y 319.986,Z 712.713,A -85,B 0,C 180,E1 -15389.483,E2 -15389.483} C_VEL
LIN {X 0,Y 319.95,Z 712.63,A -85,B 0,C 180,E1 -15392.52,E2 -15392.52} C_VEL
LIN {X 0,Y 319.901,Z 712.636,A -85,B 0,C 180,E1 -15396.308,E2 -15396.308} C_VEL
LIN {X 0,Y 319.738,Z 712.651,A -85,B 0,C 180,E1 -15400.13,E2 -15400.13} C_VEL
LIN {X 0,Y 319.736,Z 712.651,A -85,B 0,C 180,E1 -15403.994,E2 -15403.994} C_VEL
LIN {X 0,Y 319.612,Z 712.671,A -85,B 0,C 180,E1 -15407.931,E2 -15407.931} C_VEL
LIN {X 0,Y 319.568,Z 712.674,A -85,B 0,C 180,E1 -15411.956,E2 -15411.956} C_VEL
LIN {X 0,Y 319.555,Z 712.66,A -85,B 0,C 180,E1 -15416.097,E2 -15416.097} C_VEL
LIN {X 0,Y 319.53,Z 712.677,A -85,B 0,C 180,E1 -15418.941,E2 -15418.941} C_VEL
LIN {X 0,Y 319.526,Z 712.677,A -85,B 0,C 180,E1 -15421.864,E2 -15421.864} C_VEL
LIN {X 0,Y 319.584,Z 712.648,A -85,B 0,C 180,E1 -15425.543,E2 -15425.543} C_VEL
LIN {X 0,Y 319.535,Z 712.684,A -85,B 0,C 180,E1 -15429.663,E2 -15429.663} C_VEL
LIN {X 0,Y 319.516,Z 712.687,A -85,B 0,C 180,E1 -15433.459,E2 -15433.459} C_VEL
LIN {X 0,Y 319.556,Z 712.679,A -85,B 0,C 180,E1 -15437.016,E2 -15437.016} C_VEL
LIN {X 0,Y 319.505,Z 712.685,A -85,B 0,C 180,E1 -15438.669,E2 -15438.669} C_VEL
LIN {X 0,Y 318.825,Z 712.772,A -85,B 0,C 180,E1 -15439.37,E2 -15439.37} C_VEL
LIN {X 0,Y 315.979,Z 713.127,A -85,B 0,C 180,E1 -15440.47,E2 -15440.47} C_VEL
LIN {X 0,Y 313.14,Z 713.48,A -85,B 0,C 180,E1 -15441.589,E2 -15441.589} C_VEL
LIN {X 0,Y 312.497,Z 713.558,A -85,B 0,C 180,E1 -15442.312,E2 -15442.312} C_VEL
LIN {X 0,Y 312.572,Z 713.677,A -85,B 0,C 180,E1 -15443.971,E2 -15443.971} C_VEL
LIN {X 0,Y 312.773,Z 714.598,A -85,B 0,C 180,E1 -15444.197,E2 -15444.197} C_VEL
LIN {X 0,Y 320.495,Z 736.451,A -85,B 0,C 180,E1 -15445.277,E2 -15445.277} C_VEL
LIN {X 0,Y 319.158,Z 790.753,A -85,B 0,C 180,E1 -15446.825,E2 -15446.825} C_VEL
LIN {X 0,Y 318.835,Z 802.84,A -85,B 0,C 180,E1 -15447.36,E2 -15447.36} C_VEL
LIN {X 0,Y 318.49,Z 813.663,A -85,B 0,C 180,E1 -15448.021,E2 -15448.021} C_VEL
LIN {X 0,Y 317.992,Z 822.71,A -85,B 0,C 180,E1 -15448.709,E2 -15448.709} C_VEL
LIN {X 0,Y 317.313,Z 833.617,A -85,B 0,C 180,E1 -15449.748,E2 -15449.748} C_VEL
LIN {X 0,Y 316.669,Z 842.503,A -85,B 0,C 180,E1 -15450.773,E2 -15450.773} C_VEL
LIN {X 0,Y 315.971,Z 851.224,A -85,B 0,C 180,E1 -15451.973,E2 -15451.973} C_VEL
LIN {X 0,Y 315.404,Z 858.562,A -85,B 0,C 180,E1 -15453.157,E2 -15453.157} C_VEL
LIN {X 0,Y 314.778,Z 865.897,A -85,B 0,C 180,E1 -15454.545,E2 -15454.545} C_VEL
LIN {X 0,Y 314.061,Z 873.378,A -85,B 0,C 180,E1 -15456.246,E2 -15456.246} C_VEL
LIN {X 0,Y 313.587,Z 879.561,A -85,B 0,C 180,E1 -15457.951,E2 -15457.951} C_VEL
LIN {X 0,Y 313.192,Z 884.634,A -85,B 0,C 180,E1 -15459.646,E2 -15459.646} C_VEL
LIN {X 0,Y 312.883,Z 889.414,A -85,B 0,C 180,E1 -15461.671,E2 -15461.671} C_VEL
LIN {X 0,Y 312.756,Z 892.003,A -85,B 0,C 180,E1 -15463.014,E2 -15463.014} C_VEL
LIN {X 0,Y 312.679,Z 894.906,A -85,B 0,C 180,E1 -15465.134,E2 -15465.134} C_VEL
LIN {X 0,Y 312.779,Z 896.574,A -85,B 0,C 180,E1 -15467.015,E2 -15467.015} C_VEL
LIN {X 0,Y 312.965,Z 897.178,A -85,B 0,C 180,E1 -15468.34,E2 -15468.34} C_VEL
LIN {X 0,Y 313.44,Z 897.177,A -85,B 0,C 180,E1 -15470.61,E2 -15470.61} C_VEL
LIN {X 0,Y 313.879,Z 896.312,A -85,B 0,C 180,E1 -15472.279,E2 -15472.279} C_VEL
LIN {X 0,Y 314.903,Z 893.452,A -85,B 0,C 180,E1 -15474.878,E2 -15474.878} C_VEL
LIN {X 0,Y 315.804,Z 890.125,A -85,B 0,C 180,E1 -15476.81,E2 -15476.81} C_VEL
LIN {X 0,Y 316.685,Z 886.678,A -85,B 0,C 180,E1 -15478.348,E2 -15478.348} C_VEL
LIN {X 0,Y 318.02,Z 880.968,A -85,B 0,C 180,E1 -15480.316,E2 -15480.316} C_VEL
LIN {X 0,Y 319.281,Z 875.283,A -85,B 0,C 180,E1 -15481.892,E2 -15481.892} C_VEL
LIN {X 0,Y 320.62,Z 868.427,A -85,B 0,C 180,E1 -15483.456,E2 -15483.456} C_VEL
LIN {X 0,Y 321.815,Z 861.926,A -85,B 0,C 180,E1 -15484.697,E2 -15484.697} C_VEL
LIN {X 0,Y 323.216,Z 853.161,A -85,B 0,C 180,E1 -15486.085,E2 -15486.085} C_VEL
LIN {X 0,Y 324.34,Z 845.113,A -85,B 0,C 180,E1 -15487.157,E2 -15487.157} C_VEL
LIN {X 0,Y 325.484,Z 835.449,A -85,B 0,C 180,E1 -15488.224,E2 -15488.224} C_VEL
LIN {X 0,Y 326.457,Z 825.227,A -85,B 0,C 180,E1 -15489.135,E2 -15489.135} C_VEL
LIN {X 0,Y 327.161,Z 815.637,A -85,B 0,C 180,E1 -15489.817,E2 -15489.817} C_VEL
LIN {X 0,Y 327.691,Z 805.546,A -85,B 0,C 180,E1 -15490.374,E2 -15490.374} C_VEL
LIN {X 0,Y 328.022,Z 791.998,A -85,B 0,C 180,E1 -15490.922,E2 -15490.922} C_VEL
LIN {X 0,Y 329.501,Z 761.686,A -85,B 0,C 180,E1 -15491.902,E2 -15491.902} C_VEL
LIN {X 0,Y 330.413,Z 744.926,A -85,B 0,C 180,E1 -15492.447,E2 -15492.447} C_VEL
LIN {X 0,Y 325.652,Z 735.474,A -85,B 0,C 180,E1 -15493.527,E2 -15493.527} C_VEL
LIN {X 0,Y 319.977,Z 725.719,A -85,B 0,C 180,E1 -15494.885,E2 -15494.885} C_VEL
LIN {X 0,Y 317.629,Z 722.013,A -85,B 0,C 180,E1 -15495.474,E2 -15495.474} C_VEL
LIN {X 0,Y 315.159,Z 718.169,A -85,B 0,C 180,E1 -15496.124,E2 -15496.124} C_VEL
LIN {X 0,Y 313.276,Z 715.701,A -85,B 0,C 180,E1 -15496.612,E2 -15496.612} C_VEL
LIN {X 0,Y 312.687,Z 714.053,A -85,B 0,C 180,E1 -15496.913,E2 -15496.913} C_VEL
LIN {X 0,Y 312.601,Z 713.571,A -85,B 0,C 180,E1 -15497.331,E2 -15497.331} C_VEL
LIN {X 0,Y 312.542,Z 713.556,A -85,B 0,C 180,E1 -15501.087,E2 -15501.087} C_VEL
LIN {X 0,Y 312.536,Z 713.554,A -85,B 0,C 180,E1 -15503.876,E2 -15503.876} C_VEL
LIN {X 0,Y 312.516,Z 713.555,A -85,B 0,C 180,E1 -15506.729,E2 -15506.729} C_VEL
LIN {X 0,Y 312.511,Z 713.559,A -85,B 0,C 180,E1 -15509.653,E2 -15509.653} C_VEL
LIN {X 0,Y 312.527,Z 713.556,A -85,B 0,C 180,E1 -15513.688,E2 -15513.688} C_VEL
LIN {X 0,Y 312.544,Z 713.553,A -85,B 0,C 180,E1 -15517.383,E2 -15517.383} C_VEL
LIN {X 0,Y 312.497,Z 713.557,A -85,B 0,C 180,E1 -15520.708,E2 -15520.708} C_VEL
LIN {X 0,Y 312.458,Z 713.565,A -85,B 0,C 180,E1 -15524.208,E2 -15524.208} C_VEL
LIN {X 0,Y 312.49,Z 713.562,A -85,B 0,C 180,E1 -15527.917,E2 -15527.917} C_VEL
LIN {X 0,Y 312.592,Z 713.749,A -85,B 0,C 180,E1 -15531.525,E2 -15531.525} C_VEL
LIN {X 0,Y 316.028,Z 727.872,A -85,B 0,C 180,E1 -15535.101,E2 -15535.101} C_VEL
LIN {X 0,Y 319.118,Z 741.674,A -85,B 0,C 180,E1 -15538.362,E2 -15538.362} C_VEL
LIN {X 0,Y 319.723,Z 745.554,A -85,B 0,C 180,E1 -15539.237,E2 -15539.237} C_VEL
LIN {X 0,Y 318.882,Z 752.784,A -85,B 0,C 180,E1 -15540.678,E2 -15540.678} C_VEL
LIN {X 0,Y 321.188,Z 768.666,A -85,B 0,C 180,E1 -15541.798,E2 -15541.798} C_VEL
LIN {X 0,Y 323.983,Z 790.751,A -85,B 0,C 180,E1 -15543.127,E2 -15543.127} C_VEL
LIN {X 0,Y 325.485,Z 808.147,A -85,B 0,C 180,E1 -15544.031,E2 -15544.031} C_VEL
LIN {X 0,Y 326.604,Z 833.403,A -85,B 0,C 180,E1 -15545.13,E2 -15545.13} C_VEL
LIN {X 0,Y 324.274,Z 877.625,A -85,B 0,C 180,E1 -15546.53,E2 -15546.53} C_VEL
LIN {X 0,Y 323.296,Z 888.452,A -85,B 0,C 180,E1 -15547.005,E2 -15547.005} C_VEL
LIN {X 0,Y 322.114,Z 899.133,A -85,B 0,C 180,E1 -15547.636,E2 -15547.636} C_VEL
LIN {X 0,Y 320.944,Z 908.217,A -85,B 0,C 180,E1 -15548.312,E2 -15548.312} C_VEL
LIN {X 0,Y 319.703,Z 916.735,A -85,B 0,C 180,E1 -15549.068,E2 -15549.068} C_VEL
LIN {X 0,Y 318.056,Z 926.71,A -85,B 0,C 180,E1 -15550.137,E2 -15550.137} C_VEL
LIN {X 0,Y 316.456,Z 936.294,A -85,B 0,C 180,E1 -15551.381,E2 -15551.381} C_VEL
LIN {X 0,Y 315.32,Z 943.529,A -85,B 0,C 180,E1 -15552.487,E2 -15552.487} C_VEL
LIN {X 0,Y 314.046,Z 952.28,A -85,B 0,C 180,E1 -15554.087,E2 -15554.087} C_VEL
LIN {X 0,Y 313.17,Z 958.577,A -85,B 0,C 180,E1 -15555.431,E2 -15555.431} C_VEL
LIN {X 0,Y 312.034,Z 968.73,A -85,B 0,C 180,E1 -15557.973,E2 -15557.973} C_VEL
LIN {X 0,Y 311.608,Z 975.89,A -85,B 0,C 180,E1 -15560.259,E2 -15560.259} C_VEL
LIN {X 0,Y 311.542,Z 980.629,A -85,B 0,C 180,E1 -15562.219,E2 -15562.219} C_VEL
LIN {X 0,Y 311.641,Z 984.227,A -85,B 0,C 180,E1 -15564.174,E2 -15564.174} C_VEL
LIN {X 0,Y 311.929,Z 986.783,A -85,B 0,C 180,E1 -15566.122,E2 -15566.122} C_VEL
LIN {X 0,Y 311.995,Z 987.916,A -85,B 0,C 180,E1 -15567.416,E2 -15567.416} C_VEL
LIN {X 0,Y 312.102,Z 988.606,A -85,B 0,C 180,E1 -15568.708,E2 -15568.708} C_VEL
LIN {X 0,Y 312.199,Z 988.883,A -85,B 0,C 180,E1 -15569.998,E2 -15569.998} C_VEL
LIN {X 0,Y 312.085,Z 988.722,A -85,B 0,C 180,E1 -15571.288,E2 -15571.288} C_VEL
LIN {X 0,Y 311.971,Z 988.125,A -85,B 0,C 180,E1 -15572.58,E2 -15572.58} C_VEL
LIN {X 0,Y 311.92,Z 987.094,A -85,B 0,C 180,E1 -15573.874,E2 -15573.874} C_VEL
LIN {X 0,Y 311.729,Z 985.628,A -85,B 0,C 180,E1 -15575.172,E2 -15575.172} C_VEL
LIN {X 0,Y 311.555,Z 982.828,A -85,B 0,C 180,E1 -15577.001,E2 -15577.001} C_VEL
LIN {X 0,Y 311.485,Z 978.531,A -85,B 0,C 180,E1 -15579.085,E2 -15579.085} C_VEL
LIN {X 0,Y 311.728,Z 973.334,A -85,B 0,C 180,E1 -15581.046,E2 -15581.046} C_VEL
LIN {X 0,Y 312.358,Z 966.875,A -85,B 0,C 180,E1 -15583.001,E2 -15583.001} C_VEL
LIN {X 0,Y 313.293,Z 959.416,A -85,B 0,C 180,E1 -15584.834,E2 -15584.834} C_VEL
LIN {X 0,Y 314.49,Z 950.858,A -85,B 0,C 180,E1 -15586.552,E2 -15586.552} C_VEL
LIN {X 0,Y 315.917,Z 941.078,A -85,B 0,C 180,E1 -15588.144,E2 -15588.144} C_VEL
LIN {X 0,Y 317.617,Z 930.32,A -85,B 0,C 180,E1 -15589.551,E2 -15589.551} C_VEL
LIN {X 0,Y 319.307,Z 918.367,A -85,B 0,C 180,E1 -15590.786,E2 -15590.786} C_VEL
LIN {X 0,Y 320.895,Z 905.655,A -85,B 0,C 180,E1 -15591.772,E2 -15591.772} C_VEL
LIN {X 0,Y 322.246,Z 892.322,A -85,B 0,C 180,E1 -15592.519,E2 -15592.519} C_VEL
LIN {X 0,Y 323,Z 878.744,A -85,B 0,C 180,E1 -15593.013,E2 -15593.013} C_VEL
LIN {X 0,Y 324.1,Z 830.784,A -85,B 0,C 180,E1 -15594.126,E2 -15594.126} C_VEL
LIN {X 0,Y 321.336,Z 800.295,A -85,B 0,C 180,E1 -15595.131,E2 -15595.131} C_VEL
LIN {X 0,Y 317.845,Z 773.824,A -85,B 0,C 180,E1 -15596.133,E2 -15596.133} C_VEL
LIN {X 0,Y 317.311,Z 769.592,A -85,B 0,C 180,E1 -15596.336,E2 -15596.336} C_VEL
LIN {X 0,Y 320.126,Z 748.7,A -85,B 0,C 180,E1 -15600.623,E2 -15600.623} C_VEL
LIN {X 0,Y 320.116,Z 745.388,A -85,B 0,C 180,E1 -15601.357,E2 -15601.357} C_VEL
LIN {X 0,Y 317.396,Z 732.272,A -85,B 0,C 180,E1 -15604.602,E2 -15604.602} C_VEL
LIN {X 0,Y 314.502,Z 720.668,A -85,B 0,C 180,E1 -15607.712,E2 -15607.712} C_VEL
LIN {X 0,Y 312.508,Z 713.642,A -85,B 0,C 180,E1 -15609.81,E2 -15609.81} C_VEL
LIN {X 0,Y 312.473,Z 713.559,A -85,B 0,C 180,E1 -15613.968,E2 -15613.968} C_VEL
LIN {X 0,Y 312.506,Z 713.559,A -85,B 0,C 180,E1 -15617.911,E2 -15617.911} C_VEL
LIN {X 0,Y 312.526,Z 713.555,A -85,B 0,C 180,E1 -15621.909,E2 -15621.909} C_VEL
LIN {X 0,Y 312.496,Z 713.549,A -85,B 0,C 180,E1 -15625.789,E2 -15625.789} C_VEL
LIN {X 0,Y 312.514,Z 713.554,A -85,B 0,C 180,E1 -15628.853,E2 -15628.853} C_VEL
LIN {X 0,Y 312.564,Z 713.546,A -85,B 0,C 180,E1 -15631.824,E2 -15631.824} C_VEL
LIN {X 0,Y 312.574,Z 713.545,A -85,B 0,C 180,E1 -15634.71,E2 -15634.71} C_VEL
LIN {X 0,Y 312.576,Z 713.548,A -85,B 0,C 180,E1 -15637.528,E2 -15637.528} C_VEL
LIN {X 0,Y 312.627,Z 713.538,A -85,B 0,C 180,E1 -15641.656,E2 -15641.656} C_VEL
LIN {X 0,Y 312.682,Z 713.532,A -85,B 0,C 180,E1 -15645.686,E2 -15645.686} C_VEL
LIN {X 0,Y 312.686,Z 713.535,A -85,B 0,C 180,E1 -15649.641,E2 -15649.641} C_VEL
LIN {X 0,Y 312.841,Z 713.511,A -85,B 0,C 180,E1 -15652.254,E2 -15652.254} C_VEL
LIN {X 0,Y 312.705,Z 713.526,A -85,B 0,C 180,E1 -15654.842,E2 -15654.842} C_VEL
LIN {X 0,Y 312.979,Z 713.496,A -85,B 0,C 180,E1 -15658.714,E2 -15658.714} C_VEL
LIN {X 0,Y 312.979,Z 713.495,A -85,B 0,C 180,E1 -15661.287,E2 -15661.287} C_VEL
LIN {X 0,Y 312.705,Z 713.527,A -85,B 0,C 180,E1 -15665.158,E2 -15665.158} C_VEL
LIN {X 0,Y 312.86,Z 713.51,A -85,B 0,C 180,E1 -15667.746,E2 -15667.746} C_VEL
LIN {X 0,Y 312.658,Z 713.535,A -85,B 0,C 180,E1 -15671.672,E2 -15671.672} C_VEL
LIN {X 0,Y 312.689,Z 713.534,A -85,B 0,C 180,E1 -15674.888,E2 -15674.888} C_VEL
LIN {X 0,Y 312.598,Z 713.542,A -85,B 0,C 180,E1 -15679.226,E2 -15679.226} C_VEL
LIN {X 0,Y 312.515,Z 713.54,A -85,B 0,C 180,E1 -15682.781,E2 -15682.781} C_VEL
LIN {X 0,Y 312.571,Z 713.553,A -85,B 0,C 180,E1 -15686.724,E2 -15686.724} C_VEL
LIN {X 0,Y 312.528,Z 713.547,A -85,B 0,C 180,E1 -15689.652,E2 -15689.652} C_VEL
LIN {X 0,Y 312.511,Z 713.551,A -85,B 0,C 180,E1 -15693.69,E2 -15693.69} C_VEL
LIN {X 0,Y 312.53,Z 713.558,A -85,B 0,C 180,E1 -15697.385,E2 -15697.385} C_VEL
LIN {X 0,Y 312.593,Z 713.799,A -85,B 0,C 180,E1 -15698.655,E2 -15698.655} C_VEL
LIN {X 0,Y 312.85,Z 714.898,A -85,B 0,C 180,E1 -15698.87,E2 -15698.87} C_VEL
LIN {X 0,Y 322.403,Z 733.83,A -85,B 0,C 180,E1 -15700.341,E2 -15700.341} C_VEL
LIN {X 0,Y 326.008,Z 742.063,A -85,B 0,C 180,E1 -15700.888,E2 -15700.888} C_VEL
LIN {X 0,Y 325.117,Z 792.18,A -85,B 0,C 180,E1 -15702.077,E2 -15702.077} C_VEL
LIN {X 0,Y 324.986,Z 805.359,A -85,B 0,C 180,E1 -15702.534,E2 -15702.534} C_VEL
LIN {X 0,Y 324.535,Z 818.338,A -85,B 0,C 180,E1 -15703.244,E2 -15703.244} C_VEL
LIN {X 0,Y 323.821,Z 829.83,A -85,B 0,C 180,E1 -15704.107,E2 -15704.107} C_VEL
LIN {X 0,Y 322.743,Z 840.837,A -85,B 0,C 180,E1 -15705.174,E2 -15705.174} C_VEL
LIN {X 0,Y 321.477,Z 851.869,A -85,B 0,C 180,E1 -15706.542,E2 -15706.542} C_VEL
LIN {X 0,Y 320.296,Z 860.518,A -85,B 0,C 180,E1 -15707.865,E2 -15707.865} C_VEL
LIN {X 0,Y 318.968,Z 869.087,A -85,B 0,C 180,E1 -15709.462,E2 -15709.462} C_VEL
LIN {X 0,Y 317.701,Z 876.537,A -85,B 0,C 180,E1 -15711.169,E2 -15711.169} C_VEL
LIN {X 0,Y 316.46,Z 883.446,A -85,B 0,C 180,E1 -15713.16,E2 -15713.16} C_VEL
LIN {X 0,Y 315.332,Z 888.993,A -85,B 0,C 180,E1 -15715.192,E2 -15715.192} C_VEL
LIN {X 0,Y 314.37,Z 893.807,A -85,B 0,C 180,E1 -15717.554,E2 -15717.554} C_VEL
LIN {X 0,Y 313.879,Z 895.951,A -85,B 0,C 180,E1 -15719.006,E2 -15719.006} C_VEL
LIN {X 0,Y 313.442,Z 898.02,A -85,B 0,C 180,E1 -15720.982,E2 -15720.982} C_VEL
LIN {X 0,Y 313.065,Z 899.259,A -85,B 0,C 180,E1 -15723.324,E2 -15723.324} C_VEL
LIN {X 0,Y 312.945,Z 899.395,A -85,B 0,C 180,E1 -15724.744,E2 -15724.744} C_VEL
LIN {X 0,Y 312.944,Z 898.564,A -85,B 0,C 180,E1 -15727.04,E2 -15727.04} C_VEL
LIN {X 0,Y 313.163,Z 896.926,A -85,B 0,C 180,E1 -15728.959,E2 -15728.959} C_VEL
LIN {X 0,Y 313.587,Z 894.104,A -85,B 0,C 180,E1 -15731.038,E2 -15731.038} C_VEL
LIN {X 0,Y 314.211,Z 890.163,A -85,B 0,C 180,E1 -15733.098,E2 -15733.098} C_VEL
LIN {X 0,Y 314.968,Z 885.027,A -85,B 0,C 180,E1 -15735.133,E2 -15735.133} C_VEL
LIN {X 0,Y 315.905,Z 878.549,A -85,B 0,C 180,E1 -15737.148,E2 -15737.148} C_VEL
LIN {X 0,Y 316.86,Z 871.902,A -85,B 0,C 180,E1 -15738.811,E2 -15738.811} C_VEL
LIN {X 0,Y 317.936,Z 863.906,A -85,B 0,C 180,E1 -15740.459,E2 -15740.459} C_VEL
LIN {X 0,Y 319.144,Z 853.893,A -85,B 0,C 180,E1 -15742.123,E2 -15742.123} C_VEL
LIN {X 0,Y 320.278,Z 843.251,A -85,B 0,C 180,E1 -15743.545,E2 -15743.545} C_VEL
LIN {X 0,Y 321.245,Z 832.742,A -85,B 0,C 180,E1 -15744.667,E2 -15744.667} C_VEL
LIN {X 0,Y 322.069,Z 820.248,A -85,B 0,C 180,E1 -15745.7,E2 -15745.7} C_VEL
LIN {X 0,Y 322.618,Z 807.265,A -85,B 0,C 180,E1 -15746.489,E2 -15746.489} C_VEL
LIN {X 0,Y 322.815,Z 794.874,A -85,B 0,C 180,E1 -15746.999,E2 -15746.999} C_VEL
LIN {X 0,Y 323.498,Z 746.757,A -85,B 0,C 180,E1 -15748.135,E2 -15748.135} C_VEL
LIN {X 0,Y 323.592,Z 739.456,A -85,B 0,C 180,E1 -15748.306,E2 -15748.306} C_VEL
LIN {X 0,Y 315.733,Z 720.408,A -85,B 0,C 180,E1 -15749.367,E2 -15749.367} C_VEL
LIN {X 0,Y 313.153,Z 714.491,A -85,B 0,C 180,E1 -15749.749,E2 -15749.749} C_VEL
LIN {X 0,Y 312.954,Z 713.602,A -85,B 0,C 180,E1 -15750.002,E2 -15750.002} C_VEL
LIN {X 0,Y 312.899,Z 713.509,A -85,B 0,C 180,E1 -15752.577,E2 -15752.577} C_VEL
LIN {X 0,Y 312.843,Z 713.514,A -85,B 0,C 180,E1 -15756.451,E2 -15756.451} C_VEL
LIN {X 0,Y 312.755,Z 713.527,A -85,B 0,C 180,E1 -15759.052,E2 -15759.052} C_VEL
LIN {X 0,Y 312.636,Z 713.541,A -85,B 0,C 180,E1 -15762.993,E2 -15762.993} C_VEL
LIN {X 0,Y 312.626,Z 713.535,A -85,B 0,C 180,E1 -15765.652,E2 -15765.652} C_VEL
LIN {X 0,Y 312.54,Z 713.537,A -85,B 0,C 180,E1 -15769.714,E2 -15769.714} C_VEL
LIN {X 0,Y 312.523,Z 713.556,A -85,B 0,C 180,E1 -15772.778,E2 -15772.778} C_VEL
LIN {X 0,Y 312.488,Z 713.538,A -85,B 0,C 180,E1 -15776.733,E2 -15776.733} C_VEL
